REGION Network 10: HMI SpecialFuction Button Control
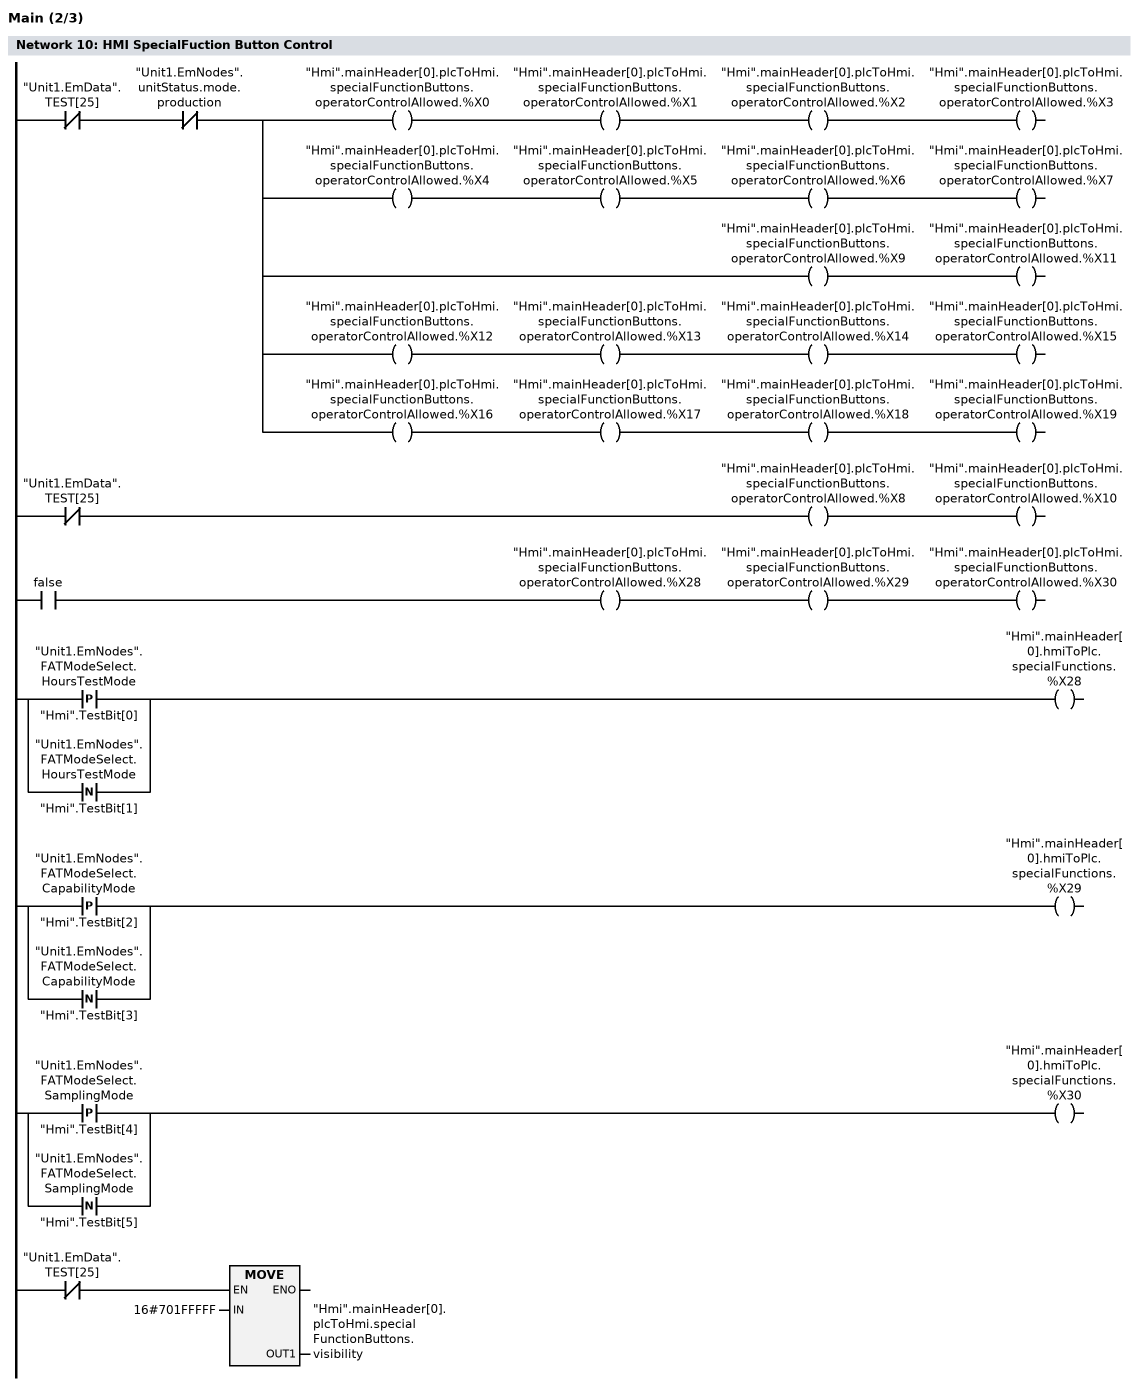
   RUNG wire#powerrail
      I_Contact( "Unit1.EmData".TEST[25] )
      I_Contact( "Unit1.EmNodes".unitStatus.mode.production )
      wire#w1
      Coil( "Hmi".mainHeader[0].plcToHmi.specialFunctionButtons.operatorControlAllowed.%X0 )
      Coil( "Hmi".mainHeader[0].plcToHmi.specialFunctionButtons.operatorControlAllowed.%X1 )
      Coil( "Hmi".mainHeader[0].plcToHmi.specialFunctionButtons.operatorControlAllowed.%X2 )
      Coil( "Hmi".mainHeader[0].plcToHmi.specialFunctionButtons.operatorControlAllowed.%X3 )
   END_RUNG
   RUNG wire#w1
      Coil( "Hmi".mainHeader[0].plcToHmi.specialFunctionButtons.operatorControlAllowed.%X4 )
      Coil( "Hmi".mainHeader[0].plcToHmi.specialFunctionButtons.operatorControlAllowed.%X5 )
      Coil( "Hmi".mainHeader[0].plcToHmi.specialFunctionButtons.operatorControlAllowed.%X6 )
      Coil( "Hmi".mainHeader[0].plcToHmi.specialFunctionButtons.operatorControlAllowed.%X7 )
   END_RUNG
   RUNG wire#w1
      Coil( "Hmi".mainHeader[0].plcToHmi.specialFunctionButtons.operatorControlAllowed.%X9 )
      Coil( "Hmi".mainHeader[0].plcToHmi.specialFunctionButtons.operatorControlAllowed.%X11 )
   END_RUNG
   RUNG wire#w1
      Coil( "Hmi".mainHeader[0].plcToHmi.specialFunctionButtons.operatorControlAllowed.%X12 )
      Coil( "Hmi".mainHeader[0].plcToHmi.specialFunctionButtons.operatorControlAllowed.%X13 )
      Coil( "Hmi".mainHeader[0].plcToHmi.specialFunctionButtons.operatorControlAllowed.%X14 )
      Coil( "Hmi".mainHeader[0].plcToHmi.specialFunctionButtons.operatorControlAllowed.%X15 )
   END_RUNG
   RUNG wire#w1
      Coil( "Hmi".mainHeader[0].plcToHmi.specialFunctionButtons.operatorControlAllowed.%X16 )
      Coil( "Hmi".mainHeader[0].plcToHmi.specialFunctionButtons.operatorControlAllowed.%X17 )
      Coil( "Hmi".mainHeader[0].plcToHmi.specialFunctionButtons.operatorControlAllowed.%X18 )
      Coil( "Hmi".mainHeader[0].plcToHmi.specialFunctionButtons.operatorControlAllowed.%X19 )
   END_RUNG
   RUNG wire#powerrail
      I_Contact( "Unit1.EmData".TEST[25] )
      Coil( "Hmi".mainHeader[0].plcToHmi.specialFunctionButtons.operatorControlAllowed.%X8 )
      Coil( "Hmi".mainHeader[0].plcToHmi.specialFunctionButtons.operatorControlAllowed.%X10 )
   END_RUNG
   RUNG wire#powerrail
      Contact( false )
      Coil( "Hmi".mainHeader[0].plcToHmi.specialFunctionButtons.operatorControlAllowed.%X28 )
      Coil( "Hmi".mainHeader[0].plcToHmi.specialFunctionButtons.operatorControlAllowed.%X29 )
      Coil( "Hmi".mainHeader[0].plcToHmi.specialFunctionButtons.operatorControlAllowed.%X30 )
   END_RUNG
   RUNG wire#powerrail
      P_Contact(operand := "Unit1.EmNodes".FATModeSelect.HoursTestMode, bit := "Hmi".TestBit[0])
      wire#w2
      Coil( "Hmi".mainHeader[0].hmiToPlc.specialFunctions.%X28 )
   END_RUNG
   RUNG wire#powerrail
      N_Contact(operand := "Unit1.EmNodes".FATModeSelect.HoursTestMode, bit := "Hmi".TestBit[1])
   END_RUNG wire#w2
   RUNG wire#powerrail
      P_Contact(operand := "Unit1.EmNodes".FATModeSelect.CapabilityMode, bit := "Hmi".TestBit[2])
      wire#w3
      Coil( "Hmi".mainHeader[0].hmiToPlc.specialFunctions.%X29 )
   END_RUNG
   RUNG wire#powerrail
      N_Contact(operand := "Unit1.EmNodes".FATModeSelect.CapabilityMode, bit := "Hmi".TestBit[3])
   END_RUNG wire#w3
   RUNG wire#powerrail
      P_Contact(operand := "Unit1.EmNodes".FATModeSelect.SamplingMode, bit := "Hmi".TestBit[4])
      wire#w4
      Coil( "Hmi".mainHeader[0].hmiToPlc.specialFunctions.%X30 )
   END_RUNG
   RUNG wire#powerrail
      N_Contact(operand := "Unit1.EmNodes".FATModeSelect.SamplingMode, bit := "Hmi".TestBit[5])
   END_RUNG wire#w4
   RUNG wire#powerrail
      I_Contact( "Unit1.EmData".TEST[25] )
      Move(in := 16#701FFFFF, out1 => "Hmi".mainHeader[0].plcToHmi.specialFunctionButtons.visibility)
   END_RUNG
   // the same network as SCL:
   "Hmi".mainHeader[0].plcToHmi.specialFunctionButtons.operatorControlAllowed.%X0 := NOT "Unit1.EmData".TEST[25] AND NOT "Unit1.EmNodes".unitStatus.mode.production;
   "Hmi".mainHeader[0].plcToHmi.specialFunctionButtons.operatorControlAllowed.%X1 := NOT "Unit1.EmData".TEST[25] AND NOT "Unit1.EmNodes".unitStatus.mode.production;
   "Hmi".mainHeader[0].plcToHmi.specialFunctionButtons.operatorControlAllowed.%X2 := NOT "Unit1.EmData".TEST[25] AND NOT "Unit1.EmNodes".unitStatus.mode.production;
   "Hmi".mainHeader[0].plcToHmi.specialFunctionButtons.operatorControlAllowed.%X3 := NOT "Unit1.EmData".TEST[25] AND NOT "Unit1.EmNodes".unitStatus.mode.production;
   "Hmi".mainHeader[0].plcToHmi.specialFunctionButtons.operatorControlAllowed.%X4 := NOT "Unit1.EmData".TEST[25] AND NOT "Unit1.EmNodes".unitStatus.mode.production;
   "Hmi".mainHeader[0].plcToHmi.specialFunctionButtons.operatorControlAllowed.%X5 := NOT "Unit1.EmData".TEST[25] AND NOT "Unit1.EmNodes".unitStatus.mode.production;
   "Hmi".mainHeader[0].plcToHmi.specialFunctionButtons.operatorControlAllowed.%X6 := NOT "Unit1.EmData".TEST[25] AND NOT "Unit1.EmNodes".unitStatus.mode.production;
   "Hmi".mainHeader[0].plcToHmi.specialFunctionButtons.operatorControlAllowed.%X7 := NOT "Unit1.EmData".TEST[25] AND NOT "Unit1.EmNodes".unitStatus.mode.production;
   "Hmi".mainHeader[0].plcToHmi.specialFunctionButtons.operatorControlAllowed.%X9 := NOT "Unit1.EmData".TEST[25] AND NOT "Unit1.EmNodes".unitStatus.mode.production;
   "Hmi".mainHeader[0].plcToHmi.specialFunctionButtons.operatorControlAllowed.%X11 := NOT "Unit1.EmData".TEST[25] AND NOT "Unit1.EmNodes".unitStatus.mode.production;
   "Hmi".mainHeader[0].plcToHmi.specialFunctionButtons.operatorControlAllowed.%X12 := NOT "Unit1.EmData".TEST[25] AND NOT "Unit1.EmNodes".unitStatus.mode.production;
   "Hmi".mainHeader[0].plcToHmi.specialFunctionButtons.operatorControlAllowed.%X13 := NOT "Unit1.EmData".TEST[25] AND NOT "Unit1.EmNodes".unitStatus.mode.production;
   "Hmi".mainHeader[0].plcToHmi.specialFunctionButtons.operatorControlAllowed.%X14 := NOT "Unit1.EmData".TEST[25] AND NOT "Unit1.EmNodes".unitStatus.mode.production;
   "Hmi".mainHeader[0].plcToHmi.specialFunctionButtons.operatorControlAllowed.%X15 := NOT "Unit1.EmData".TEST[25] AND NOT "Unit1.EmNodes".unitStatus.mode.production;
   "Hmi".mainHeader[0].plcToHmi.specialFunctionButtons.operatorControlAllowed.%X16 := NOT "Unit1.EmData".TEST[25] AND NOT "Unit1.EmNodes".unitStatus.mode.production;
   "Hmi".mainHeader[0].plcToHmi.specialFunctionButtons.operatorControlAllowed.%X17 := NOT "Unit1.EmData".TEST[25] AND NOT "Unit1.EmNodes".unitStatus.mode.production;
   "Hmi".mainHeader[0].plcToHmi.specialFunctionButtons.operatorControlAllowed.%X18 := NOT "Unit1.EmData".TEST[25] AND NOT "Unit1.EmNodes".unitStatus.mode.production;
   "Hmi".mainHeader[0].plcToHmi.specialFunctionButtons.operatorControlAllowed.%X19 := NOT "Unit1.EmData".TEST[25] AND NOT "Unit1.EmNodes".unitStatus.mode.production;
   "Hmi".mainHeader[0].plcToHmi.specialFunctionButtons.operatorControlAllowed.%X8 := NOT "Unit1.EmData".TEST[25];
   "Hmi".mainHeader[0].plcToHmi.specialFunctionButtons.operatorControlAllowed.%X10 := NOT "Unit1.EmData".TEST[25];
   "Hmi".mainHeader[0].plcToHmi.specialFunctionButtons.operatorControlAllowed.%X28 := false;
   "Hmi".mainHeader[0].plcToHmi.specialFunctionButtons.operatorControlAllowed.%X29 := false;
   "Hmi".mainHeader[0].plcToHmi.specialFunctionButtons.operatorControlAllowed.%X30 := false;
   #_w1 := "Unit1.EmNodes".FATModeSelect.HoursTestMode AND NOT "Hmi".TestBit[0];   // rising edge of "Unit1.EmNodes".FATModeSelect.HoursTestMode
   "Hmi".TestBit[0] := "Unit1.EmNodes".FATModeSelect.HoursTestMode;
   #_w2 := NOT "Unit1.EmNodes".FATModeSelect.HoursTestMode AND "Hmi".TestBit[1];   // falling edge of "Unit1.EmNodes".FATModeSelect.HoursTestMode
   "Hmi".TestBit[1] := "Unit1.EmNodes".FATModeSelect.HoursTestMode;
   "Hmi".mainHeader[0].hmiToPlc.specialFunctions.%X28 := #_w1 OR #_w2;
   #_w3 := "Unit1.EmNodes".FATModeSelect.CapabilityMode AND NOT "Hmi".TestBit[2];   // rising edge of "Unit1.EmNodes".FATModeSelect.CapabilityMode
   "Hmi".TestBit[2] := "Unit1.EmNodes".FATModeSelect.CapabilityMode;
   #_w4 := NOT "Unit1.EmNodes".FATModeSelect.CapabilityMode AND "Hmi".TestBit[3];   // falling edge of "Unit1.EmNodes".FATModeSelect.CapabilityMode
   "Hmi".TestBit[3] := "Unit1.EmNodes".FATModeSelect.CapabilityMode;
   "Hmi".mainHeader[0].hmiToPlc.specialFunctions.%X29 := #_w3 OR #_w4;
   #_w5 := "Unit1.EmNodes".FATModeSelect.SamplingMode AND NOT "Hmi".TestBit[4];   // rising edge of "Unit1.EmNodes".FATModeSelect.SamplingMode
   "Hmi".TestBit[4] := "Unit1.EmNodes".FATModeSelect.SamplingMode;
   #_w6 := NOT "Unit1.EmNodes".FATModeSelect.SamplingMode AND "Hmi".TestBit[5];   // falling edge of "Unit1.EmNodes".FATModeSelect.SamplingMode
   "Hmi".TestBit[5] := "Unit1.EmNodes".FATModeSelect.SamplingMode;
   "Hmi".mainHeader[0].hmiToPlc.specialFunctions.%X30 := #_w5 OR #_w6;
   IF NOT "Unit1.EmData".TEST[25] THEN
       "Hmi".mainHeader[0].plcToHmi.specialFunctionButtons.visibility := 16#701FFFFF;
   END_IF;
END_REGION

REGION Network 11
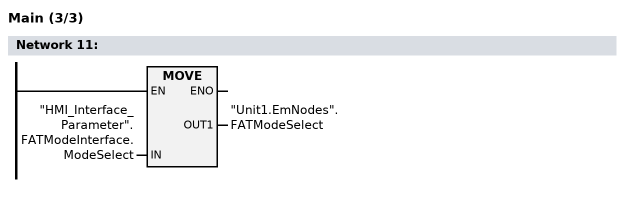
   RUNG wire#powerrail
      Move(in := "HMI_Interface_Parameter".FATModeInterface.ModeSelect, out1 => "Unit1.EmNodes".FATModeSelect)
   END_RUNG
   // the same network as SCL:
   "Unit1.EmNodes".FATModeSelect := "HMI_Interface_Parameter".FATModeInterface.ModeSelect;
END_REGION
END_ORGANIZATION_BLOCK

FUNCTION_BLOCK "CallGlobal"   // FB48, LAD
TITLE = CallGlobal
// All blocks that provide data to the DB Global.Data are called here. That includes blocks to generate system data as well as blocks that connect handle multiple HMIs.
// stored: IsIECCheckEnabled true, MemoryReserve 100, SetENOAutomatically true
   VAR
      statClockSysMemOld { ExternalWritable := 'False'} : Byte;   // Old value system memory evaluation
      statTonTimer : Array[0..10] of IEC_TIMER;
      instLAF_PowerOnOff { ExternalWritable := 'False'} : "LAF_PowerOnOff";
      instLAF_HmiHeaderManager { ExternalWritable := 'False'} : "LAF_HmiHeaderManager";
      instLAF_ClockGen { ExternalWritable := 'False'} : "LAF_ClockGenerator";
      instLSNTP_Server { ExternalWritable := 'False'} : "LSNTP_Server";
      instRemoteAccess { ExternalWritable := 'False'} : "LRemoteAccess_MobilePanelMonitor";
      statPulse : Array[0..99] of Bool;
   END_VAR
   VAR_TEMP
      tempIndex : DInt;   // Temp variable for for loop
      tempAcknowledge : Bool;   // Summarized acknowledge command
      tempPowerOff : Bool;   // Summarized power off command
      tempPowerOn : Bool;   // Summarized power on command
      tempPowerStatus : Int;   // 0 - Off, 1 - Paused, 2 - On
      tempResultXor : Byte;   // Interim result of XOR operation
      tempPosPulse : Byte;   // Interim result puls calculation
   END_VAR
   VAR CONSTANT
      RESET_BUTTON__COULD_BE_ADDED_HERE : Bool := false;   // Placeholder for a potential global reset button
      TRUE : Bool := true;
   END_VAR
   VAR_TEMP   // added for the SCL form of the ladder/FBD networks
      _w1 : Bool;
      _w2 : Bool;
      _w3 : Bool;
   END_VAR
BEGIN

REGION Network 1 (SCL): Summarize HMI commands
   // Read commands for acknowledge, powerOn and powerOff from the different HMI panels and summarize them in temp variables for further logic in this block.
   // Initialize temp variables
   #tempAcknowledge :=
   #tempPowerOff :=
   #tempPowerOn := FALSE;

   // Loop through the HMI panels and summarize the commands
   FOR #tempIndex := 0 TO "NO_OF_PANELS" DO
       #tempAcknowledge := #tempAcknowledge OR "Hmi".mainHeader[#tempIndex].hmiToPlc.acknowledge;
       #tempPowerOff := #tempPowerOff OR "Hmi".mainHeader[#tempIndex].hmiToPlc.powerCommands.%X0;
       #tempPowerOn := #tempPowerOn OR "Hmi".mainHeader[#tempIndex].hmiToPlc.powerCommands.%X1;
   END_FOR;
END_REGION

REGION Network 2: Global Acknowledge
   // The global acknowledge command from the hmi button is assigned to Global.Data.general.acknowledge: This bit it forwarded to all underlaying modules
   // If a hard-wired global reset button exists, it can
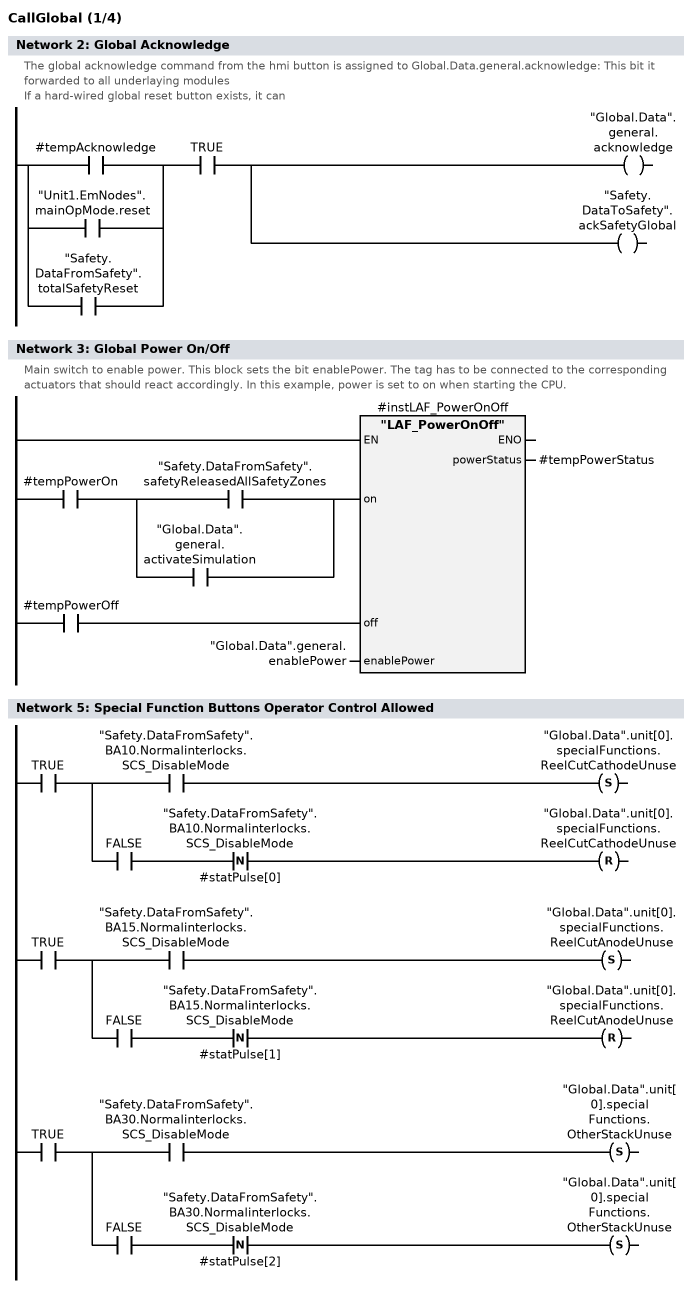
   RUNG wire#powerrail
      Contact( #tempAcknowledge )
      wire#w1
      Contact( TRUE )
      wire#w2
      Coil( "Global.Data".general.acknowledge )
   END_RUNG
   RUNG wire#powerrail
      Contact( "Unit1.EmNodes".mainOpMode.reset )
   END_RUNG wire#w1
   RUNG wire#powerrail
      Contact( "Safety.DataFromSafety".totalSafetyReset )
   END_RUNG wire#w1
   RUNG wire#w2
      Coil( "Safety.DataToSafety".ackSafetyGlobal )
   END_RUNG
   // the same network as SCL:
   "Global.Data".general.acknowledge := (#tempAcknowledge OR "Unit1.EmNodes".mainOpMode.reset OR "Safety.DataFromSafety".totalSafetyReset) AND TRUE;
   "Safety.DataToSafety".ackSafetyGlobal := "Global.Data".general.acknowledge;
END_REGION

REGION Network 3: Global Power On/Off
   // Main switch to enable power. This block sets the bit enablePower. The tag has to be connected to the corresponding actuators that should react accordingly. In this example, power is set to on when starting the CPU.
   RUNG wire#powerrail
      #instLAF_PowerOnOff(on := wire#w2, off := wire#w3, enablePower := "Global.Data".general.enablePower, powerStatus => #tempPowerStatus)
   END_RUNG
   RUNG wire#powerrail
      Contact( #tempPowerOn )
      wire#w1
      Contact( "Safety.DataFromSafety".safetyReleasedAllSafetyZones )
   END_RUNG wire#w2
   RUNG wire#w1
      Contact( "Global.Data".general.activateSimulation )
   END_RUNG wire#w2
   RUNG wire#powerrail
      Contact( #tempPowerOff )
   END_RUNG wire#w3
   // the same network as SCL:
   #instLAF_PowerOnOff(on := #tempPowerOn AND ("Safety.DataFromSafety".safetyReleasedAllSafetyZones OR "Global.Data".general.activateSimulation),   // "LAF_PowerOnOff"
                       off := #tempPowerOff,
                       enablePower := "Global.Data".general.enablePower,
                       powerStatus => #tempPowerStatus);
END_REGION

REGION Network 4 (SCL): Write power status to HMI panels
   // Write power status back to all connected HMI panels
   // Loop through the panels and set the power status
   FOR #tempIndex := 0 TO "NO_OF_PANELS" DO
       "Hmi".mainHeader[#tempIndex].plcToHmi.powerStatus := #tempPowerStatus;
   END_FOR;
END_REGION

REGION Network 5: Special Function Buttons Operator Control Allowed
   RUNG wire#powerrail
      Contact( TRUE )
      wire#w1
      Contact( "Safety.DataFromSafety".BA10.Normalinterlocks.SCS_DisableMode )
      S_Coil( "Global.Data".unit[0].specialFunctions.ReelCutCathodeUnuse )
   END_RUNG
   RUNG wire#w1
      Contact( FALSE )
      N_Contact(operand := "Safety.DataFromSafety".BA10.Normalinterlocks.SCS_DisableMode, bit := #statPulse[0])
      R_Coil( "Global.Data".unit[0].specialFunctions.ReelCutCathodeUnuse )
   END_RUNG
   RUNG wire#powerrail
      Contact( TRUE )
      wire#w2
      Contact( "Safety.DataFromSafety".BA15.Normalinterlocks.SCS_DisableMode )
      S_Coil( "Global.Data".unit[0].specialFunctions.ReelCutAnodeUnuse )
   END_RUNG
   RUNG wire#w2
      Contact( FALSE )
      N_Contact(operand := "Safety.DataFromSafety".BA15.Normalinterlocks.SCS_DisableMode, bit := #statPulse[1])
      R_Coil( "Global.Data".unit[0].specialFunctions.ReelCutAnodeUnuse )
   END_RUNG
   RUNG wire#powerrail
      Contact( TRUE )
      wire#w3
      Contact( "Safety.DataFromSafety".BA30.Normalinterlocks.SCS_DisableMode )
      S_Coil( "Global.Data".unit[0].specialFunctions.OtherStackUnuse )
   END_RUNG
   RUNG wire#w3
      Contact( FALSE )
      N_Contact(operand := "Safety.DataFromSafety".BA30.Normalinterlocks.SCS_DisableMode, bit := #statPulse[2])
      S_Coil( "Global.Data".unit[0].specialFunctions.OtherStackUnuse )
   END_RUNG
   // the same network as SCL:
   IF TRUE AND "Safety.DataFromSafety".BA10.Normalinterlocks.SCS_DisableMode THEN
       "Global.Data".unit[0].specialFunctions.ReelCutCathodeUnuse := TRUE;
   END_IF;
   #_w1 := TRUE AND FALSE AND NOT "Safety.DataFromSafety".BA10.Normalinterlocks.SCS_DisableMode AND #statPulse[0];   // falling edge of "Safety.DataFromSafety".BA10.Normalinterlocks.SCS_DisableMode
   #statPulse[0] := "Safety.DataFromSafety".BA10.Normalinterlocks.SCS_DisableMode;
   IF #_w1 THEN "Global.Data".unit[0].specialFunctions.ReelCutCathodeUnuse := FALSE; END_IF;
   IF TRUE AND "Safety.DataFromSafety".BA15.Normalinterlocks.SCS_DisableMode THEN
       "Global.Data".unit[0].specialFunctions.ReelCutAnodeUnuse := TRUE;
   END_IF;
   #_w2 := TRUE AND FALSE AND NOT "Safety.DataFromSafety".BA15.Normalinterlocks.SCS_DisableMode AND #statPulse[1];   // falling edge of "Safety.DataFromSafety".BA15.Normalinterlocks.SCS_DisableMode
   #statPulse[1] := "Safety.DataFromSafety".BA15.Normalinterlocks.SCS_DisableMode;
   IF #_w2 THEN "Global.Data".unit[0].specialFunctions.ReelCutAnodeUnuse := FALSE; END_IF;
   IF TRUE AND "Safety.DataFromSafety".BA30.Normalinterlocks.SCS_DisableMode THEN
       "Global.Data".unit[0].specialFunctions.OtherStackUnuse := TRUE;
   END_IF;
   #_w3 := TRUE AND FALSE AND NOT "Safety.DataFromSafety".BA30.Normalinterlocks.SCS_DisableMode AND #statPulse[2];   // falling edge of "Safety.DataFromSafety".BA30.Normalinterlocks.SCS_DisableMode
   #statPulse[2] := "Safety.DataFromSafety".BA30.Normalinterlocks.SCS_DisableMode;
   IF #_w3 THEN "Global.Data".unit[0].specialFunctions.OtherStackUnuse := TRUE; END_IF;
END_REGION

REGION Network 6: HMI Control Header
   // Read the input from the control header in the HMI an distribute information to the according units. Vice versa, summarize the unit information and provide it to the control header to display e.g. the modes and states.
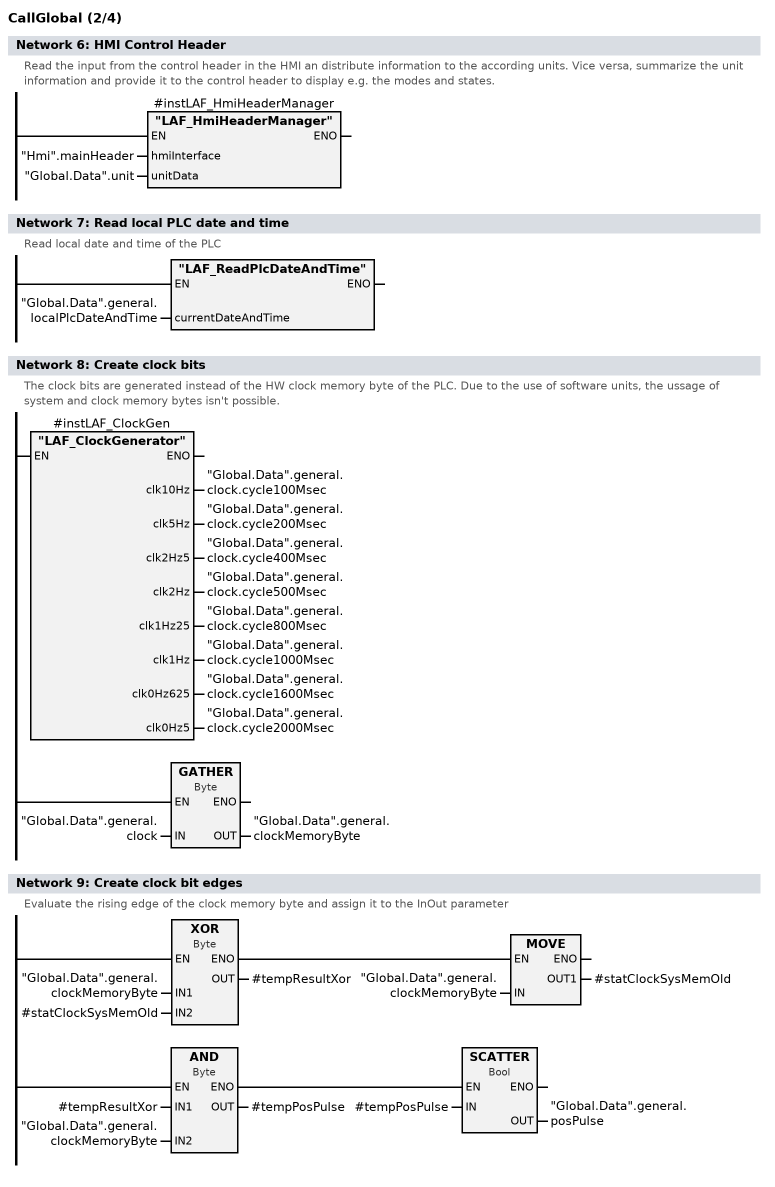
   RUNG wire#powerrail
      #instLAF_HmiHeaderManager(hmiInterface := "Hmi".mainHeader, unitData := "Global.Data".unit)
   END_RUNG
   // the same network as SCL:
   #instLAF_HmiHeaderManager(hmiInterface := "Hmi".mainHeader, unitData := "Global.Data".unit);   // "LAF_HmiHeaderManager"
END_REGION

REGION Network 7: Read local PLC date and time
   // Read local date and time of the PLC
   RUNG wire#powerrail
      "LAF_ReadPlcDateAndTime"(currentDateAndTime := "Global.Data".general.localPlcDateAndTime)
   END_RUNG
   // the same network as SCL:
   "LAF_ReadPlcDateAndTime"(currentDateAndTime := "Global.Data".general.localPlcDateAndTime);
END_REGION

REGION Network 8: Create clock bits
   // The clock bits are generated instead of the HW clock memory byte of the PLC. Due to the use of software units, the ussage of system and clock memory bytes isn't possible.
   RUNG wire#powerrail
      #instLAF_ClockGen(clk10Hz => "Global.Data".general.clock.cycle100Msec, clk5Hz => "Global.Data".general.clock.cycle200Msec, clk2Hz5 => "Global.Data".general.clock.cycle400Msec, clk2Hz => "Global.Data".general.clock.cycle500Msec, clk1Hz25 => "Global.Data".general.clock.cycle800Msec, clk1Hz => "Global.Data".general.clock.cycle1000Msec, clk0Hz625 => "Global.Data".general.clock.cycle1600Msec, clk0Hz5 => "Global.Data".general.clock.cycle2000Msec)
   END_RUNG
   RUNG wire#powerrail
      { S7_Templates := "[dest_type := Byte, src_type := Bool]" } GATHER(IN := "Global.Data".general.clock, OUT => "Global.Data".general.clockMemoryByte)
   END_RUNG
   // the same network as SCL:
   #instLAF_ClockGen(clk10Hz => "Global.Data".general.clock.cycle100Msec,   // "LAF_ClockGenerator"
                     clk5Hz => "Global.Data".general.clock.cycle200Msec,
                     clk2Hz5 => "Global.Data".general.clock.cycle400Msec,
                     clk2Hz => "Global.Data".general.clock.cycle500Msec,
                     clk1Hz25 => "Global.Data".general.clock.cycle800Msec,
                     clk1Hz => "Global.Data".general.clock.cycle1000Msec,
                     clk0Hz625 => "Global.Data".general.clock.cycle1600Msec,
                     clk0Hz5 => "Global.Data".general.clock.cycle2000Msec);
   GATHER(IN := "Global.Data".general.clock, OUT => "Global.Data".general.clockMemoryByte);
END_REGION

REGION Network 9: Create clock bit edges
   // Evaluate the rising edge of the clock memory byte and assign it to the InOut parameter
   #tempResultXor := "Global.Data".general.clockMemoryByte XOR #statClockSysMemOld;
   #statClockSysMemOld := "Global.Data".general.clockMemoryByte;
   #tempPosPulse := #tempResultXor AND "Global.Data".general.clockMemoryByte;
   SCATTER(IN := #tempPosPulse, OUT => "Global.Data".general.posPulse);
END_REGION

REGION Network 10: Time Synchronisation (NTP)
   // With the LSNTP_Server block, the NTP server will be enabled on S7 PLC, to wich the NTP client (e.g. Panel), can synchronize their data and time.
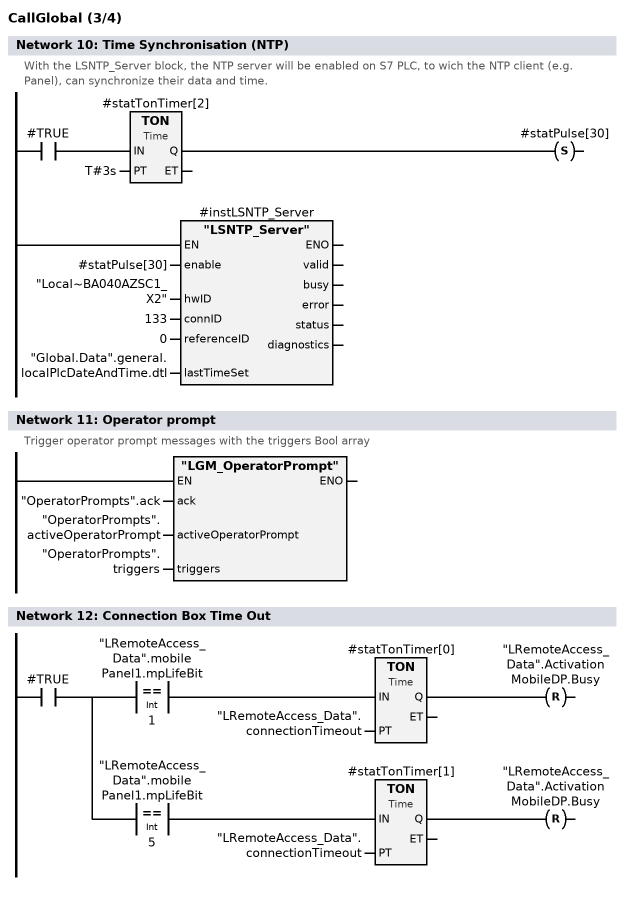
   RUNG wire#powerrail
      Contact( #TRUE )
      { S7_Templates := "time_type := Time" } #statTonTimer[2].TON(pt := T#3s, et =>)
      S_Coil( #statPulse[30] )
   END_RUNG
   RUNG wire#powerrail
      #instLSNTP_Server(enable := #statPulse[30], hwID := "Local~BA040AZSC1_X2", connID := 133, referenceID := 0, lastTimeSet := "Global.Data".general.localPlcDateAndTime.dtl, valid =>, busy =>, error =>, status =>, diagnostics =>)
   END_RUNG
   // the same network as SCL:
   #statTonTimer[2].TON(IN := #TRUE, PT := T#3s);
   IF #statTonTimer[2].Q THEN #statPulse[30] := TRUE; END_IF;
   #instLSNTP_Server(enable := #statPulse[30],   // "LSNTP_Server"
                     hwID := "Local~BA040AZSC1_X2",
                     connID := 133,
                     referenceID := 0,
                     lastTimeSet := "Global.Data".general.localPlcDateAndTime.dtl);
END_REGION

REGION Network 11: Operator prompt
   // Trigger operator prompt messages with the triggers Bool array
   RUNG wire#powerrail
      "LGM_OperatorPrompt"(ack := "OperatorPrompts".ack, activeOperatorPrompt := "OperatorPrompts".activeOperatorPrompt, triggers := "OperatorPrompts".triggers)
   END_RUNG
   // the same network as SCL:
   "LGM_OperatorPrompt"(ack := "OperatorPrompts".ack,
                        activeOperatorPrompt := "OperatorPrompts".activeOperatorPrompt,
                        triggers := "OperatorPrompts".triggers);
END_REGION

REGION Network 12: Connection Box Time Out
   RUNG wire#powerrail
      Contact( #TRUE )
      wire#w1
      { S7_Templates := "SrcType := Int" } EQ_Contact(in1 := "LRemoteAccess_Data".mobilePanel1.mpLifeBit, in2 := 1)
      { S7_Templates := "time_type := Time" } #statTonTimer[0].TON(pt := "LRemoteAccess_Data".connectionTimeout, et =>)
      R_Coil( "LRemoteAccess_Data".ActivationMobileDP.Busy )
   END_RUNG
   RUNG wire#w1
      { S7_Templates := "SrcType := Int" } EQ_Contact(in1 := "LRemoteAccess_Data".mobilePanel1.mpLifeBit, in2 := 5)
      { S7_Templates := "time_type := Time" } #statTonTimer[1].TON(pt := "LRemoteAccess_Data".connectionTimeout, et =>)
      R_Coil( "LRemoteAccess_Data".ActivationMobileDP.Busy )
   END_RUNG
   // the same network as SCL:
   #statTonTimer[0].TON(IN := #TRUE AND ("LRemoteAccess_Data".mobilePanel1.mpLifeBit = 1),
                        PT := "LRemoteAccess_Data".connectionTimeout);
   IF #statTonTimer[0].Q THEN "LRemoteAccess_Data".ActivationMobileDP.Busy := FALSE; END_IF;
   #statTonTimer[1].TON(IN := #TRUE AND ("LRemoteAccess_Data".mobilePanel1.mpLifeBit = 5),
                        PT := "LRemoteAccess_Data".connectionTimeout);
   IF #statTonTimer[1].Q THEN "LRemoteAccess_Data".ActivationMobileDP.Busy := FALSE; END_IF;
END_REGION

REGION Network 13: Connection box is connected
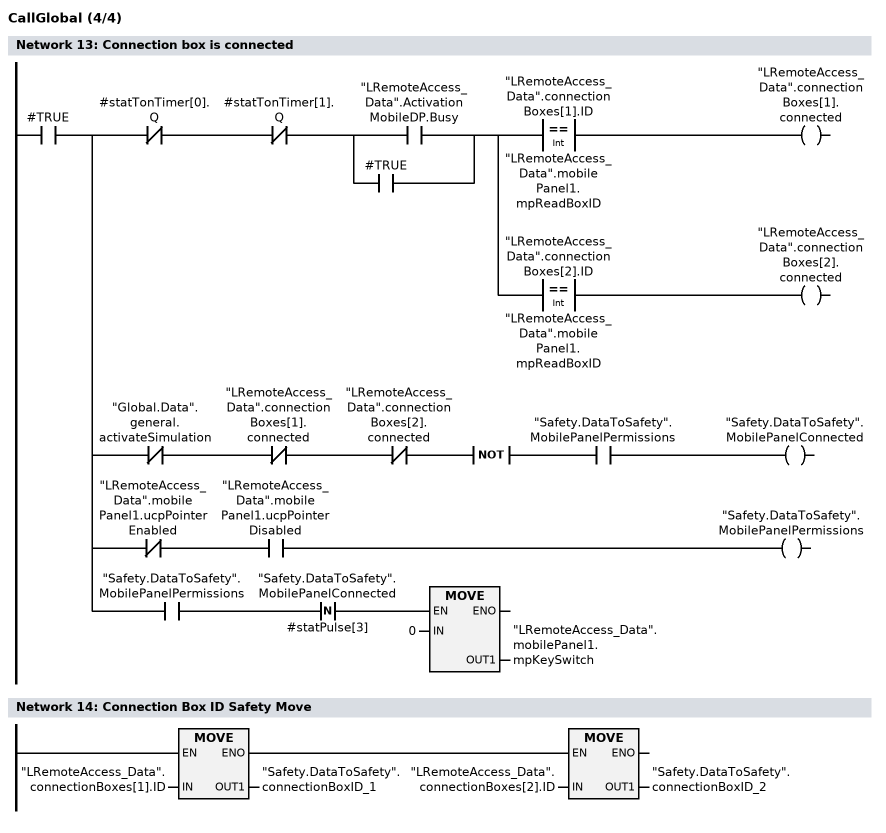
   RUNG wire#powerrail
      Contact( #TRUE )
      wire#w1
      I_Contact( #statTonTimer[0].Q )
      I_Contact( #statTonTimer[1].Q )
      wire#w2
      Contact( "LRemoteAccess_Data".ActivationMobileDP.Busy )
      wire#w3
      { S7_Templates := "SrcType := Int" } EQ_Contact(in1 := "LRemoteAccess_Data".connectionBoxes[1].ID, in2 := "LRemoteAccess_Data".mobilePanel1.mpReadBoxID)
      Coil( "LRemoteAccess_Data".connectionBoxes[1].connected )
   END_RUNG
   RUNG wire#w2
      Contact( #TRUE )
   END_RUNG wire#w3
   RUNG wire#w3
      { S7_Templates := "SrcType := Int" } EQ_Contact(in1 := "LRemoteAccess_Data".connectionBoxes[2].ID, in2 := "LRemoteAccess_Data".mobilePanel1.mpReadBoxID)
      Coil( "LRemoteAccess_Data".connectionBoxes[2].connected )
   END_RUNG
   RUNG wire#w1
      I_Contact( "Global.Data".general.activateSimulation )
      I_Contact( "LRemoteAccess_Data".connectionBoxes[1].connected )
      I_Contact( "LRemoteAccess_Data".connectionBoxes[2].connected )
      Not()
      Contact( "Safety.DataToSafety".MobilePanelPermissions )
      Coil( "Safety.DataToSafety".MobilePanelConnected )
   END_RUNG
   RUNG wire#w1
      I_Contact( "LRemoteAccess_Data".mobilePanel1.ucpPointerEnabled )
      Contact( "LRemoteAccess_Data".mobilePanel1.ucpPointerDisabled )
      Coil( "Safety.DataToSafety".MobilePanelPermissions )
   END_RUNG
   RUNG wire#w1
      Contact( "Safety.DataToSafety".MobilePanelPermissions )
      N_Contact(operand := "Safety.DataToSafety".MobilePanelConnected, bit := #statPulse[3])
      Move(in := 0, out1 => "LRemoteAccess_Data".mobilePanel1.mpKeySwitch)
   END_RUNG
   // the same network as SCL:
   #_w1 := #TRUE AND NOT #statTonTimer[0].Q AND NOT #statTonTimer[1].Q AND ("LRemoteAccess_Data".ActivationMobileDP.Busy OR #TRUE);
   "LRemoteAccess_Data".connectionBoxes[1].connected := #_w1 AND ("LRemoteAccess_Data".connectionBoxes[1].ID = "LRemoteAccess_Data".mobilePanel1.mpReadBoxID);
   "LRemoteAccess_Data".connectionBoxes[2].connected := #_w1 AND ("LRemoteAccess_Data".connectionBoxes[2].ID = "LRemoteAccess_Data".mobilePanel1.mpReadBoxID);
   "Safety.DataToSafety".MobilePanelConnected := NOT (#TRUE AND NOT "Global.Data".general.activateSimulation AND NOT "LRemoteAccess_Data".connectionBoxes[1].connected AND NOT "LRemoteAccess_Data".connectionBoxes[2].connected) AND "Safety.DataToSafety".MobilePanelPermissions;
   "Safety.DataToSafety".MobilePanelPermissions := #TRUE AND NOT "LRemoteAccess_Data".mobilePanel1.ucpPointerEnabled AND "LRemoteAccess_Data".mobilePanel1.ucpPointerDisabled;
   #_w2 := #TRUE AND "Safety.DataToSafety".MobilePanelPermissions AND NOT "Safety.DataToSafety".MobilePanelConnected AND #statPulse[3];   // falling edge of "Safety.DataToSafety".MobilePanelConnected
   #statPulse[3] := "Safety.DataToSafety".MobilePanelConnected;
   IF #_w2 THEN "LRemoteAccess_Data".mobilePanel1.mpKeySwitch := 0; END_IF;
END_REGION

REGION Network 14: Connection Box ID Safety Move
   RUNG wire#powerrail
      Move(in := "LRemoteAccess_Data".connectionBoxes[1].ID, out1 => "Safety.DataToSafety".connectionBoxID_1)
      Move(in := "LRemoteAccess_Data".connectionBoxes[2].ID, out1 => "Safety.DataToSafety".connectionBoxID_2)
   END_RUNG
   // the same network as SCL:
   "Safety.DataToSafety".connectionBoxID_1 := "LRemoteAccess_Data".connectionBoxes[1].ID;
   "Safety.DataToSafety".connectionBoxID_2 := "LRemoteAccess_Data".connectionBoxes[2].ID;
END_REGION
END_FUNCTION_BLOCK

FUNCTION_BLOCK "CallSimulation"   // FB19, LAD
// stored: MemoryReserve 100, SetENOAutomatically false
   VAR
      instSimRotaryAxis { ExternalAccessible := 'False'; ExternalVisible := 'False'; ExternalWritable := 'False'} : Array[0..49] of "LER_SimHmiRotaryAxis";
      Unwindwe1 { S7_SetPoint := 'True'} : "LER_SimHmiRotaryAxis";
      IEC_Timer_0_Instance { S7_SetPoint := 'True'} : TON_TIME;
      "LER_SimAxis+_Axis07_pnp1X" { S7_SetPoint := 'True'} : "LER_SimAxis+";
      "LER_SimAxis+_Axis10_pnp1Z" { S7_SetPoint := 'True'} : "LER_SimAxis+";
      "LER_SimAxis+_Axis8_pnp2X" { S7_SetPoint := 'True'} : "LER_SimAxis+";
      "LER_SimAxis+_Axis13_pnp2Z" { S7_SetPoint := 'True'} : "LER_SimAxis+";
      "LER_SimAxis+_Axis12_pnp1Z" { S7_SetPoint := 'True'} : "LER_SimAxis+";
      "LER_SimAxis+_Axis14_pnp2Z" { S7_SetPoint := 'True'} : "LER_SimAxis+";
      "LER_SimAxis+_Axis34_cutterX" { S7_SetPoint := 'True'} : "LER_SimAxis+";
      "LER_SimAxis+_Axis35_cutterZ" { S7_SetPoint := 'True'} : "LER_SimAxis+";
      "LER_SimAxis-_Axis36_GripperX" { S7_SetPoint := 'True'} : "LER_SimAxis-";
      "LER_SimAxis+_Axis37_gripperZ" { S7_SetPoint := 'True'} : "LER_SimAxis+";
      "LER_SimAxis-_Axis32_StackTableZ" { S7_SetPoint := 'True'} : "LER_SimAxis-";
      "LER_SimAxis+_Axis21_roller" { S7_SetPoint := 'True'} : "LER_SimAxis+";
      "LER_SimAxis+_gripperAxis_C" { S7_SetPoint := 'True'} : "LER_SimAxis+";
      IEC_Timer_1_Instance { S7_SetPoint := 'True'} : TON_TIME;
      "LER_SimAxis+_Axis05_pnp1X" { S7_SetPoint := 'True'} : "LER_SimAxis+";
      "LER_SimAxis+_Axis06_pnp2X" { S7_SetPoint := 'True'} : "LER_SimAxis+";
   END_VAR
   VAR CONSTANT
      FALSE : Bool := FALSE;
      TRUE : Bool := TRUE;
   END_VAR
   VAR_TEMP   // added for the SCL form of the ladder/FBD networks
      _w1 : Bool;
      _w2 : Bool;
      _w3 : Bool;
      _w4 : Bool;
      _w5 : Bool;
      _w6 : Bool;
      _w7 : Bool;
      _w8 : Bool;
   END_VAR
BEGIN

REGION Network 1: SIMIT simulation currently running
   // The input "0.000CC1-KE50_I1.6_SimitRunning" is a life bit from SIMIT, which is always TRUE while SIMIT is running. The following actions are performed in that case:
   // - Simulation button in HMI is not shown when a SIMIT simulation is currently running
   // - Deactivate PLC internal simulation while SIMIT simulation is running
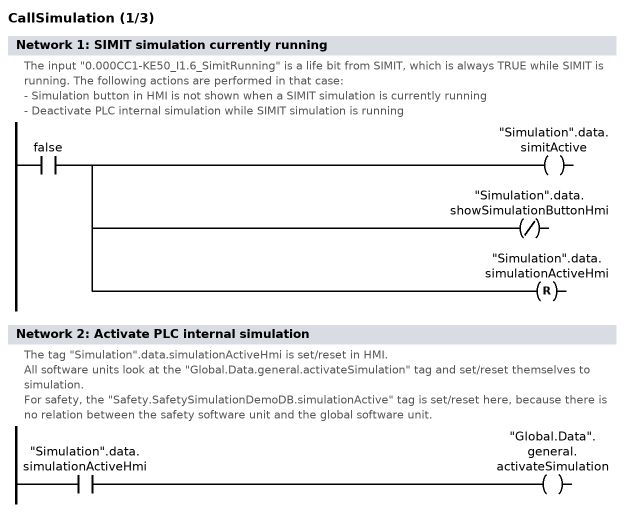
   RUNG wire#powerrail
      Contact( false )
      wire#w1
      Coil( "Simulation".data.simitActive )
   END_RUNG
   RUNG wire#w1
      I_Coil( "Simulation".data.showSimulationButtonHmi )
   END_RUNG
   RUNG wire#w1
      R_Coil( "Simulation".data.simulationActiveHmi )
   END_RUNG
   // the same network as SCL:
   "Simulation".data.simitActive := false;
   "Simulation".data.showSimulationButtonHmi := NOT false;
   IF false THEN "Simulation".data.simulationActiveHmi := FALSE; END_IF;
END_REGION

REGION Network 2: Activate PLC internal simulation
   // The tag "Simulation".data.simulationActiveHmi is set/reset in HMI.
   // 
   // All software units look at the "Global.Data.general.activateSimulation" tag and set/reset themselves to simulation.
   // 
   // For safety, the "Safety.SafetySimulationDemoDB.simulationActive" tag is set/reset here, because there is no relation between the safety software unit and the global software unit.
   RUNG wire#powerrail
      Contact( "Simulation".data.simulationActiveHmi )
      Coil( "Global.Data".general.activateSimulation )
   END_RUNG
   // the same network as SCL:
   "Global.Data".general.activateSimulation := "Simulation".data.simulationActiveHmi;
END_REGION

REGION Network 3: Simulation Linear Axis
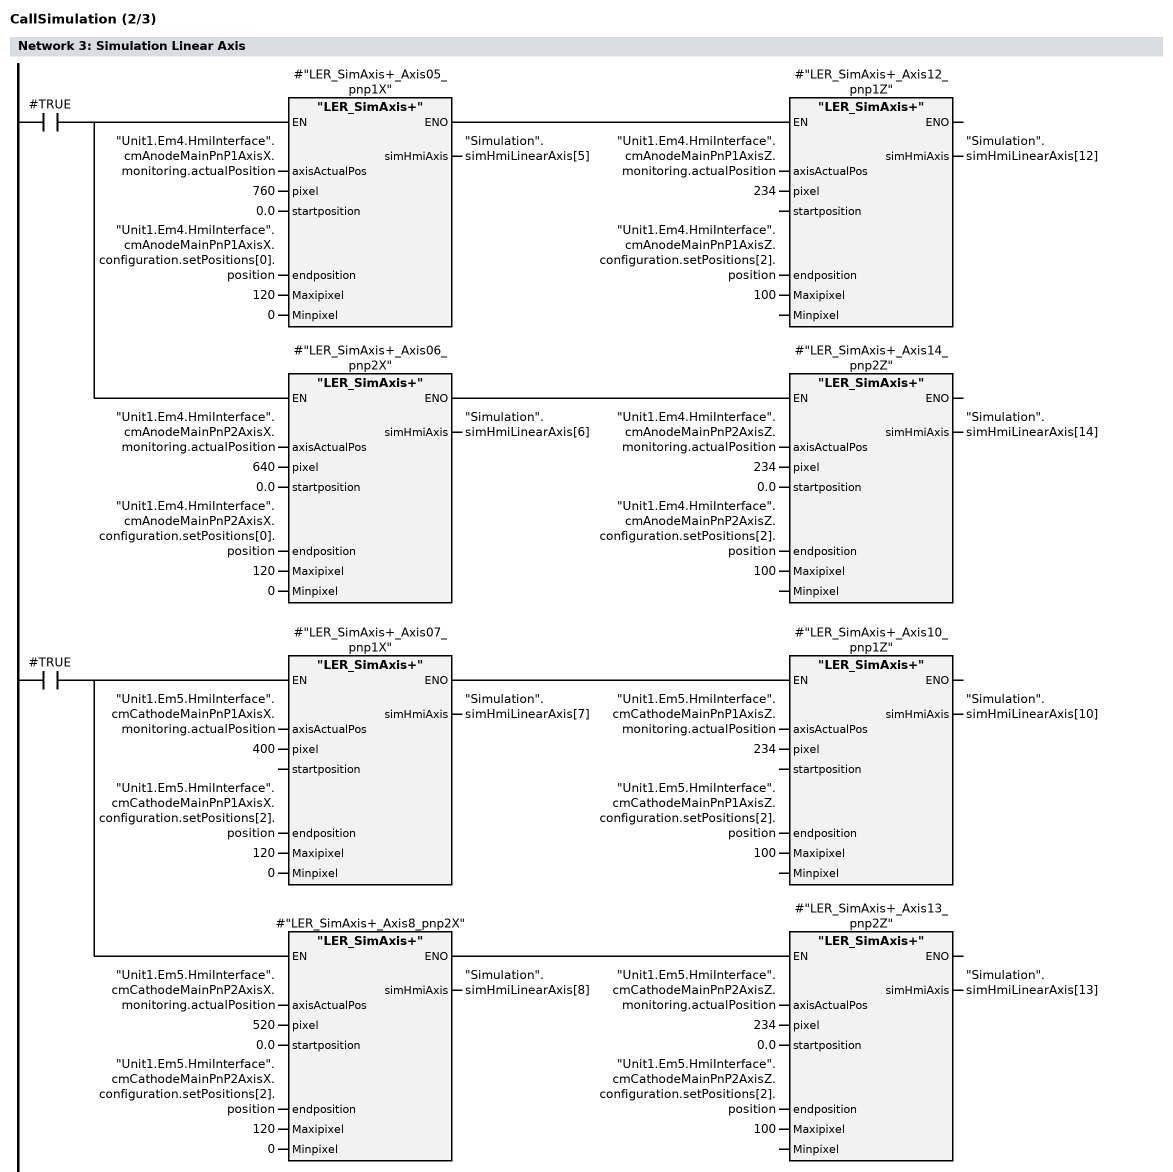
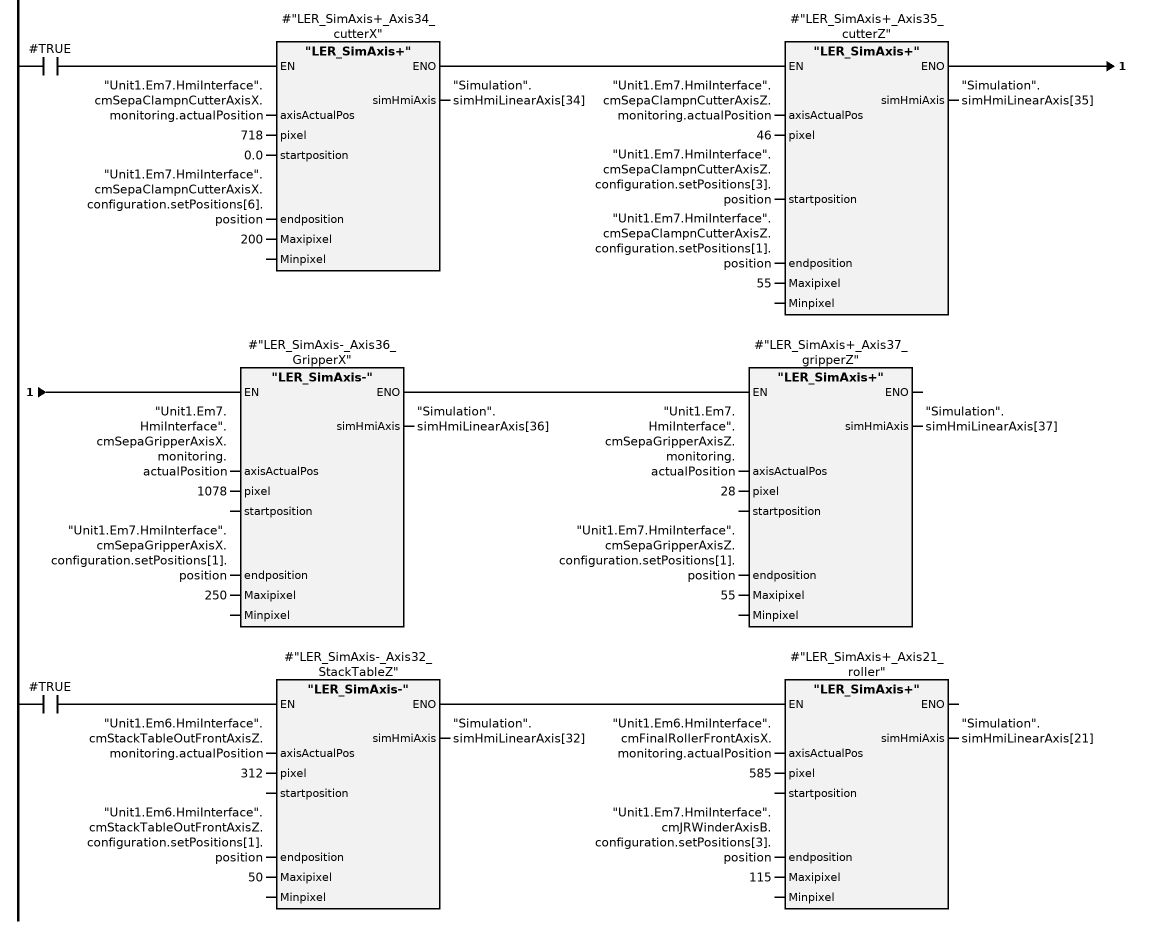
   RUNG wire#powerrail
      Contact( #TRUE )
      wire#w1
      #"LER_SimAxis+_Axis05_pnp1X"(axisActualPos := "Unit1.Em4.HmiInterface".cmAnodeMainPnP1AxisX.monitoring.actualPosition, pixel := 760, startposition := 0.0, endposition := "Unit1.Em4.HmiInterface".cmAnodeMainPnP1AxisX.configuration.setPositions[0].position, Maxipixel := 120, Minpixel := 0, simHmiAxis => "Simulation".simHmiLinearAxis[5])
      #"LER_SimAxis+_Axis12_pnp1Z"(axisActualPos := "Unit1.Em4.HmiInterface".cmAnodeMainPnP1AxisZ.monitoring.actualPosition, pixel := 234, startposition :=, endposition := "Unit1.Em4.HmiInterface".cmAnodeMainPnP1AxisZ.configuration.setPositions[2].position, Maxipixel := 100, Minpixel :=, simHmiAxis => "Simulation".simHmiLinearAxis[12])
   END_RUNG
   RUNG wire#w1
      #"LER_SimAxis+_Axis06_pnp2X"(axisActualPos := "Unit1.Em4.HmiInterface".cmAnodeMainPnP2AxisX.monitoring.actualPosition, pixel := 640, startposition := 0.0, endposition := "Unit1.Em4.HmiInterface".cmAnodeMainPnP2AxisX.configuration.setPositions[0].position, Maxipixel := 120, Minpixel := 0, simHmiAxis => "Simulation".simHmiLinearAxis[6])
      #"LER_SimAxis+_Axis14_pnp2Z"(axisActualPos := "Unit1.Em4.HmiInterface".cmAnodeMainPnP2AxisZ.monitoring.actualPosition, pixel := 234, startposition := 0.0, endposition := "Unit1.Em4.HmiInterface".cmAnodeMainPnP2AxisZ.configuration.setPositions[2].position, Maxipixel := 100, Minpixel :=, simHmiAxis => "Simulation".simHmiLinearAxis[14])
   END_RUNG
   RUNG wire#powerrail
      Contact( #TRUE )
      wire#w2
      #"LER_SimAxis+_Axis07_pnp1X"(axisActualPos := "Unit1.Em5.HmiInterface".cmCathodeMainPnP1AxisX.monitoring.actualPosition, pixel := 400, startposition :=, endposition := "Unit1.Em5.HmiInterface".cmCathodeMainPnP1AxisX.configuration.setPositions[2].position, Maxipixel := 120, Minpixel := 0, simHmiAxis => "Simulation".simHmiLinearAxis[7])
      #"LER_SimAxis+_Axis10_pnp1Z"(axisActualPos := "Unit1.Em5.HmiInterface".cmCathodeMainPnP1AxisZ.monitoring.actualPosition, pixel := 234, startposition :=, endposition := "Unit1.Em5.HmiInterface".cmCathodeMainPnP1AxisZ.configuration.setPositions[2].position, Maxipixel := 100, Minpixel :=, simHmiAxis => "Simulation".simHmiLinearAxis[10])
   END_RUNG
   RUNG wire#w2
      #"LER_SimAxis+_Axis8_pnp2X"(axisActualPos := "Unit1.Em5.HmiInterface".cmCathodeMainPnP2AxisX.monitoring.actualPosition, pixel := 520, startposition := 0.0, endposition := "Unit1.Em5.HmiInterface".cmCathodeMainPnP2AxisX.configuration.setPositions[2].position, Maxipixel := 120, Minpixel := 0, simHmiAxis => "Simulation".simHmiLinearAxis[8])
      #"LER_SimAxis+_Axis13_pnp2Z"(axisActualPos := "Unit1.Em5.HmiInterface".cmCathodeMainPnP2AxisZ.monitoring.actualPosition, pixel := 234, startposition := 0.0, endposition := "Unit1.Em5.HmiInterface".cmCathodeMainPnP2AxisZ.configuration.setPositions[2].position, Maxipixel := 100, Minpixel :=, simHmiAxis => "Simulation".simHmiLinearAxis[13])
   END_RUNG
   RUNG wire#powerrail
      Contact( #TRUE )
      #"LER_SimAxis+_Axis34_cutterX"(axisActualPos := "Unit1.Em7.HmiInterface".cmSepaClampnCutterAxisX.monitoring.actualPosition, pixel := 718, startposition := 0.0, endposition := "Unit1.Em7.HmiInterface".cmSepaClampnCutterAxisX.configuration.setPositions[6].position, Maxipixel := 200, Minpixel :=, simHmiAxis => "Simulation".simHmiLinearAxis[34])
      #"LER_SimAxis+_Axis35_cutterZ"(axisActualPos := "Unit1.Em7.HmiInterface".cmSepaClampnCutterAxisZ.monitoring.actualPosition, pixel := 46, startposition := "Unit1.Em7.HmiInterface".cmSepaClampnCutterAxisZ.configuration.setPositions[3].position, endposition := "Unit1.Em7.HmiInterface".cmSepaClampnCutterAxisZ.configuration.setPositions[1].position, Maxipixel := 55, Minpixel :=, simHmiAxis => "Simulation".simHmiLinearAxis[35])
      #"LER_SimAxis-_Axis36_GripperX"(axisActualPos := "Unit1.Em7.HmiInterface".cmSepaGripperAxisX.monitoring.actualPosition, pixel := 1078, startposition :=, endposition := "Unit1.Em7.HmiInterface".cmSepaGripperAxisX.configuration.setPositions[1].position, Maxipixel := 250, Minpixel :=, simHmiAxis => "Simulation".simHmiLinearAxis[36])
      #"LER_SimAxis+_Axis37_gripperZ"(axisActualPos := "Unit1.Em7.HmiInterface".cmSepaGripperAxisZ.monitoring.actualPosition, pixel := 28, startposition :=, endposition := "Unit1.Em7.HmiInterface".cmSepaGripperAxisZ.configuration.setPositions[1].position, Maxipixel := 55, Minpixel :=, simHmiAxis => "Simulation".simHmiLinearAxis[37])
   END_RUNG
   RUNG wire#powerrail
      Contact( #TRUE )
      #"LER_SimAxis-_Axis32_StackTableZ"(axisActualPos := "Unit1.Em6.HmiInterface".cmStackTableOutFrontAxisZ.monitoring.actualPosition, pixel := 312, startposition :=, endposition := "Unit1.Em6.HmiInterface".cmStackTableOutFrontAxisZ.configuration.setPositions[1].position, Maxipixel := 50, Minpixel :=, simHmiAxis => "Simulation".simHmiLinearAxis[32])
      #"LER_SimAxis+_Axis21_roller"(axisActualPos := "Unit1.Em6.HmiInterface".cmFinalRollerFrontAxisX.monitoring.actualPosition, pixel := 585, startposition :=, endposition := "Unit1.Em7.HmiInterface".cmJRWinderAxisB.configuration.setPositions[3].position, Maxipixel := 115, Minpixel :=, simHmiAxis => "Simulation".simHmiLinearAxis[21])
   END_RUNG
   // the same network as SCL:
   #"LER_SimAxis+_Axis05_pnp1X"(EN := #TRUE,   // "LER_SimAxis+"
                           axisActualPos := "Unit1.Em4.HmiInterface".cmAnodeMainPnP1AxisX.monitoring.actualPosition,
                           pixel := 760,
                           startposition := 0.0,
                           endposition := "Unit1.Em4.HmiInterface".cmAnodeMainPnP1AxisX.configuration.setPositions[0].position,
                           Maxipixel := 120,
                           Minpixel := 0,
                           simHmiAxis => "Simulation".simHmiLinearAxis[5],
                           ENO => #_w1);
   IF #_w1 THEN
       #"LER_SimAxis+_Axis12_pnp1Z"(axisActualPos := "Unit1.Em4.HmiInterface".cmAnodeMainPnP1AxisZ.monitoring.actualPosition,   // "LER_SimAxis+"
                               pixel := 234,
                               endposition := "Unit1.Em4.HmiInterface".cmAnodeMainPnP1AxisZ.configuration.setPositions[2].position,
                               Maxipixel := 100,
                               simHmiAxis => "Simulation".simHmiLinearAxis[12]);
   END_IF;
   #"LER_SimAxis+_Axis06_pnp2X"(EN := #TRUE,   // "LER_SimAxis+"
                           axisActualPos := "Unit1.Em4.HmiInterface".cmAnodeMainPnP2AxisX.monitoring.actualPosition,
                           pixel := 640,
                           startposition := 0.0,
                           endposition := "Unit1.Em4.HmiInterface".cmAnodeMainPnP2AxisX.configuration.setPositions[0].position,
                           Maxipixel := 120,
                           Minpixel := 0,
                           simHmiAxis => "Simulation".simHmiLinearAxis[6],
                           ENO => #_w2);
   IF #_w2 THEN
       #"LER_SimAxis+_Axis14_pnp2Z"(axisActualPos := "Unit1.Em4.HmiInterface".cmAnodeMainPnP2AxisZ.monitoring.actualPosition,   // "LER_SimAxis+"
                               pixel := 234,
                               startposition := 0.0,
                               endposition := "Unit1.Em4.HmiInterface".cmAnodeMainPnP2AxisZ.configuration.setPositions[2].position,
                               Maxipixel := 100,
                               simHmiAxis => "Simulation".simHmiLinearAxis[14]);
   END_IF;
   #"LER_SimAxis+_Axis07_pnp1X"(EN := #TRUE,   // "LER_SimAxis+"
                           axisActualPos := "Unit1.Em5.HmiInterface".cmCathodeMainPnP1AxisX.monitoring.actualPosition,
                           pixel := 400,
                           endposition := "Unit1.Em5.HmiInterface".cmCathodeMainPnP1AxisX.configuration.setPositions[2].position,
                           Maxipixel := 120,
                           Minpixel := 0,
                           simHmiAxis => "Simulation".simHmiLinearAxis[7],
                           ENO => #_w3);
   IF #_w3 THEN
       #"LER_SimAxis+_Axis10_pnp1Z"(axisActualPos := "Unit1.Em5.HmiInterface".cmCathodeMainPnP1AxisZ.monitoring.actualPosition,   // "LER_SimAxis+"
                               pixel := 234,
                               endposition := "Unit1.Em5.HmiInterface".cmCathodeMainPnP1AxisZ.configuration.setPositions[2].position,
                               Maxipixel := 100,
                               simHmiAxis => "Simulation".simHmiLinearAxis[10]);
   END_IF;
   #"LER_SimAxis+_Axis8_pnp2X"(EN := #TRUE,   // "LER_SimAxis+"
                           axisActualPos := "Unit1.Em5.HmiInterface".cmCathodeMainPnP2AxisX.monitoring.actualPosition,
                           pixel := 520,
                           startposition := 0.0,
                           endposition := "Unit1.Em5.HmiInterface".cmCathodeMainPnP2AxisX.configuration.setPositions[2].position,
                           Maxipixel := 120,
                           Minpixel := 0,
                           simHmiAxis => "Simulation".simHmiLinearAxis[8],
                           ENO => #_w4);
   IF #_w4 THEN
       #"LER_SimAxis+_Axis13_pnp2Z"(axisActualPos := "Unit1.Em5.HmiInterface".cmCathodeMainPnP2AxisZ.monitoring.actualPosition,   // "LER_SimAxis+"
                               pixel := 234,
                               startposition := 0.0,
                               endposition := "Unit1.Em5.HmiInterface".cmCathodeMainPnP2AxisZ.configuration.setPositions[2].position,
                               Maxipixel := 100,
                               simHmiAxis => "Simulation".simHmiLinearAxis[13]);
   END_IF;
   #"LER_SimAxis+_Axis34_cutterX"(EN := #TRUE,   // "LER_SimAxis+"
                           axisActualPos := "Unit1.Em7.HmiInterface".cmSepaClampnCutterAxisX.monitoring.actualPosition,
                           pixel := 718,
                           startposition := 0.0,
                           endposition := "Unit1.Em7.HmiInterface".cmSepaClampnCutterAxisX.configuration.setPositions[6].position,
                           Maxipixel := 200,
                           simHmiAxis => "Simulation".simHmiLinearAxis[34],
                           ENO => #_w5);
   #"LER_SimAxis+_Axis35_cutterZ"(EN := #_w5,   // "LER_SimAxis+"
                           axisActualPos := "Unit1.Em7.HmiInterface".cmSepaClampnCutterAxisZ.monitoring.actualPosition,
                           pixel := 46,
                           startposition := "Unit1.Em7.HmiInterface".cmSepaClampnCutterAxisZ.configuration.setPositions[3].position,
                           endposition := "Unit1.Em7.HmiInterface".cmSepaClampnCutterAxisZ.configuration.setPositions[1].position,
                           Maxipixel := 55,
                           simHmiAxis => "Simulation".simHmiLinearAxis[35],
                           ENO => #_w6);
   #"LER_SimAxis-_Axis36_GripperX"(EN := #_w6,   // "LER_SimAxis-"
                           axisActualPos := "Unit1.Em7.HmiInterface".cmSepaGripperAxisX.monitoring.actualPosition,
                           pixel := 1078,
                           endposition := "Unit1.Em7.HmiInterface".cmSepaGripperAxisX.configuration.setPositions[1].position,
                           Maxipixel := 250,
                           simHmiAxis => "Simulation".simHmiLinearAxis[36],
                           ENO => #_w7);
   IF #_w7 THEN
       #"LER_SimAxis+_Axis37_gripperZ"(axisActualPos := "Unit1.Em7.HmiInterface".cmSepaGripperAxisZ.monitoring.actualPosition,   // "LER_SimAxis+"
                               pixel := 28,
                               endposition := "Unit1.Em7.HmiInterface".cmSepaGripperAxisZ.configuration.setPositions[1].position,
                               Maxipixel := 55,
                               simHmiAxis => "Simulation".simHmiLinearAxis[37]);
   END_IF;
   #"LER_SimAxis-_Axis32_StackTableZ"(EN := #TRUE,   // "LER_SimAxis-"
                           axisActualPos := "Unit1.Em6.HmiInterface".cmStackTableOutFrontAxisZ.monitoring.actualPosition,
                           pixel := 312,
                           endposition := "Unit1.Em6.HmiInterface".cmStackTableOutFrontAxisZ.configuration.setPositions[1].position,
                           Maxipixel := 50,
                           simHmiAxis => "Simulation".simHmiLinearAxis[32],
                           ENO => #_w8);
   IF #_w8 THEN
       #"LER_SimAxis+_Axis21_roller"(axisActualPos := "Unit1.Em6.HmiInterface".cmFinalRollerFrontAxisX.monitoring.actualPosition,   // "LER_SimAxis+"
                               pixel := 585,
                               endposition := "Unit1.Em7.HmiInterface".cmJRWinderAxisB.configuration.setPositions[3].position,
                               Maxipixel := 115,
                               simHmiAxis => "Simulation".simHmiLinearAxis[21]);
   END_IF;
END_REGION

REGION Network 4: Simulation Rotary Axis
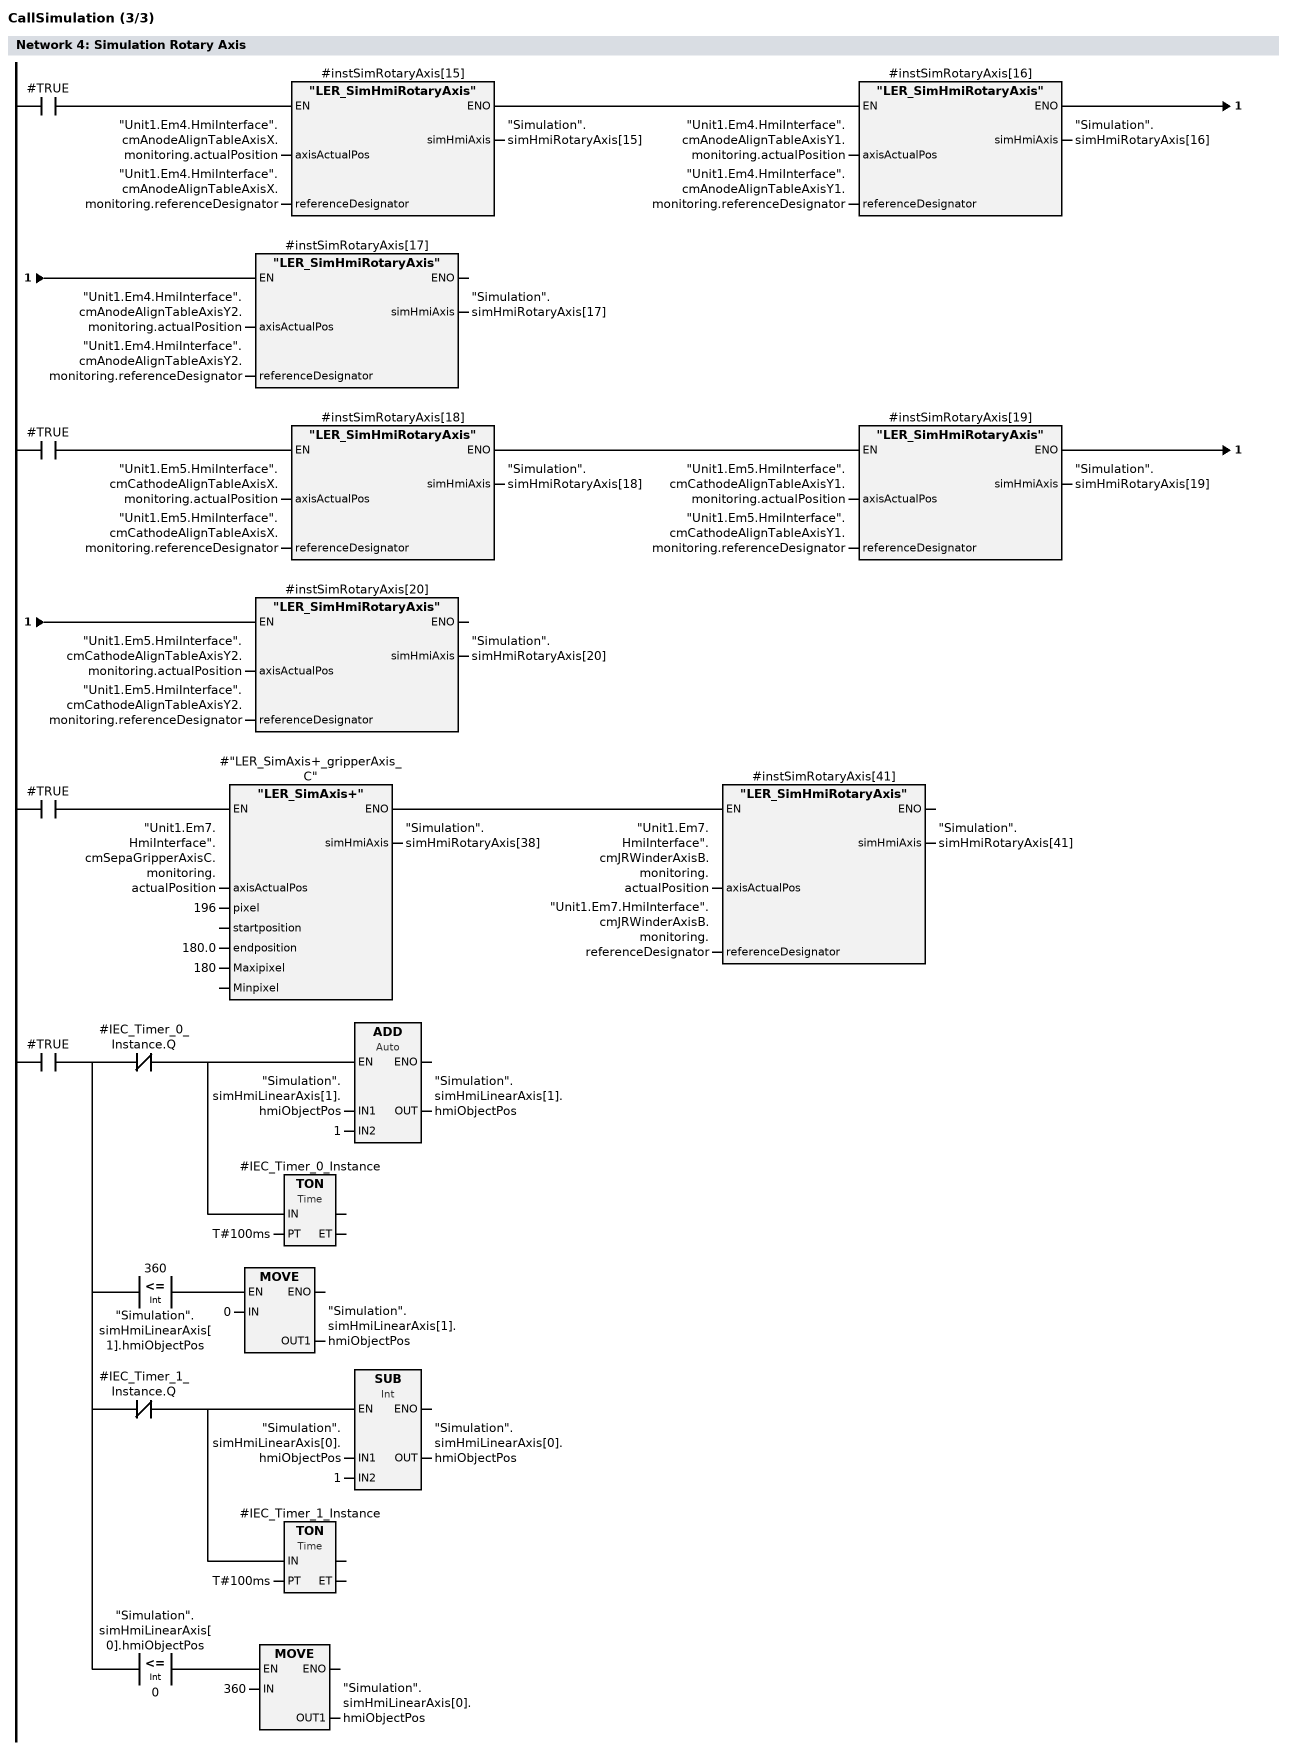
   RUNG wire#powerrail
      Contact( #TRUE )
      #instSimRotaryAxis[15](axisActualPos := "Unit1.Em4.HmiInterface".cmAnodeAlignTableAxisX.monitoring.actualPosition, referenceDesignator := "Unit1.Em4.HmiInterface".cmAnodeAlignTableAxisX.monitoring.referenceDesignator, simHmiAxis => "Simulation".simHmiRotaryAxis[15])
      #instSimRotaryAxis[16](axisActualPos := "Unit1.Em4.HmiInterface".cmAnodeAlignTableAxisY1.monitoring.actualPosition, referenceDesignator := "Unit1.Em4.HmiInterface".cmAnodeAlignTableAxisY1.monitoring.referenceDesignator, simHmiAxis => "Simulation".simHmiRotaryAxis[16])
      #instSimRotaryAxis[17](axisActualPos := "Unit1.Em4.HmiInterface".cmAnodeAlignTableAxisY2.monitoring.actualPosition, referenceDesignator := "Unit1.Em4.HmiInterface".cmAnodeAlignTableAxisY2.monitoring.referenceDesignator, simHmiAxis => "Simulation".simHmiRotaryAxis[17])
   END_RUNG
   RUNG wire#powerrail
      Contact( #TRUE )
      #instSimRotaryAxis[18](axisActualPos := "Unit1.Em5.HmiInterface".cmCathodeAlignTableAxisX.monitoring.actualPosition, referenceDesignator := "Unit1.Em5.HmiInterface".cmCathodeAlignTableAxisX.monitoring.referenceDesignator, simHmiAxis => "Simulation".simHmiRotaryAxis[18])
      #instSimRotaryAxis[19](axisActualPos := "Unit1.Em5.HmiInterface".cmCathodeAlignTableAxisY1.monitoring.actualPosition, referenceDesignator := "Unit1.Em5.HmiInterface".cmCathodeAlignTableAxisY1.monitoring.referenceDesignator, simHmiAxis => "Simulation".simHmiRotaryAxis[19])
      #instSimRotaryAxis[20](axisActualPos := "Unit1.Em5.HmiInterface".cmCathodeAlignTableAxisY2.monitoring.actualPosition, referenceDesignator := "Unit1.Em5.HmiInterface".cmCathodeAlignTableAxisY2.monitoring.referenceDesignator, simHmiAxis => "Simulation".simHmiRotaryAxis[20])
   END_RUNG
   RUNG wire#powerrail
      Contact( #TRUE )
      #"LER_SimAxis+_gripperAxis_C"(axisActualPos := "Unit1.Em7.HmiInterface".cmSepaGripperAxisC.monitoring.actualPosition, pixel := 196, startposition :=, endposition := 180.0, Maxipixel := 180, Minpixel :=, simHmiAxis => "Simulation".simHmiRotaryAxis[38])
      #instSimRotaryAxis[41](axisActualPos := "Unit1.Em7.HmiInterface".cmJRWinderAxisB.monitoring.actualPosition, referenceDesignator := "Unit1.Em7.HmiInterface".cmJRWinderAxisB.monitoring.referenceDesignator, simHmiAxis => "Simulation".simHmiRotaryAxis[41])
   END_RUNG
   RUNG wire#powerrail
      Contact( #TRUE )
      wire#w1
      I_Contact( #IEC_Timer_0_Instance.Q )
      wire#w2
      Add(in1 := "Simulation".simHmiLinearAxis[1].hmiObjectPos, in2 := 1, out => "Simulation".simHmiLinearAxis[1].hmiObjectPos)
   END_RUNG
   RUNG wire#w2
      { S7_Templates := "time_type := Time" } #IEC_Timer_0_Instance.TON(pt := T#100ms, et =>)
   END_RUNG
   RUNG wire#w1
      { S7_Templates := "SrcType := Int" } LE_Contact(in1 := 360, in2 := "Simulation".simHmiLinearAxis[1].hmiObjectPos)
      Move(in := 0, out1 => "Simulation".simHmiLinearAxis[1].hmiObjectPos)
   END_RUNG
   RUNG wire#w1
      I_Contact( #IEC_Timer_1_Instance.Q )
      wire#w3
      { S7_Templates := "SrcType := Int" } Sub(in1 := "Simulation".simHmiLinearAxis[0].hmiObjectPos, in2 := 1, out => "Simulation".simHmiLinearAxis[0].hmiObjectPos)
   END_RUNG
   RUNG wire#w3
      { S7_Templates := "time_type := Time" } #IEC_Timer_1_Instance.TON(pt := T#100ms, et =>)
   END_RUNG
   RUNG wire#w1
      { S7_Templates := "SrcType := Int" } LE_Contact(in1 := "Simulation".simHmiLinearAxis[0].hmiObjectPos, in2 := 0)
      Move(in := 360, out1 => "Simulation".simHmiLinearAxis[0].hmiObjectPos)
   END_RUNG
   // the same network as SCL:
   #instSimRotaryAxis[15](EN := #TRUE,   // "LER_SimHmiRotaryAxis"
                          axisActualPos := "Unit1.Em4.HmiInterface".cmAnodeAlignTableAxisX.monitoring.actualPosition,
                          referenceDesignator := "Unit1.Em4.HmiInterface".cmAnodeAlignTableAxisX.monitoring.referenceDesignator,
                          simHmiAxis => "Simulation".simHmiRotaryAxis[15],
                          ENO => #_w1);
   #instSimRotaryAxis[16](EN := #_w1,   // "LER_SimHmiRotaryAxis"
                          axisActualPos := "Unit1.Em4.HmiInterface".cmAnodeAlignTableAxisY1.monitoring.actualPosition,
                          referenceDesignator := "Unit1.Em4.HmiInterface".cmAnodeAlignTableAxisY1.monitoring.referenceDesignator,
                          simHmiAxis => "Simulation".simHmiRotaryAxis[16],
                          ENO => #_w2);
   IF #_w2 THEN
       #instSimRotaryAxis[17](axisActualPos := "Unit1.Em4.HmiInterface".cmAnodeAlignTableAxisY2.monitoring.actualPosition,   // "LER_SimHmiRotaryAxis"
                              referenceDesignator := "Unit1.Em4.HmiInterface".cmAnodeAlignTableAxisY2.monitoring.referenceDesignator,
                              simHmiAxis => "Simulation".simHmiRotaryAxis[17]);
   END_IF;
   #instSimRotaryAxis[18](EN := #TRUE,   // "LER_SimHmiRotaryAxis"
                          axisActualPos := "Unit1.Em5.HmiInterface".cmCathodeAlignTableAxisX.monitoring.actualPosition,
                          referenceDesignator := "Unit1.Em5.HmiInterface".cmCathodeAlignTableAxisX.monitoring.referenceDesignator,
                          simHmiAxis => "Simulation".simHmiRotaryAxis[18],
                          ENO => #_w3);
   #instSimRotaryAxis[19](EN := #_w3,   // "LER_SimHmiRotaryAxis"
                          axisActualPos := "Unit1.Em5.HmiInterface".cmCathodeAlignTableAxisY1.monitoring.actualPosition,
                          referenceDesignator := "Unit1.Em5.HmiInterface".cmCathodeAlignTableAxisY1.monitoring.referenceDesignator,
                          simHmiAxis => "Simulation".simHmiRotaryAxis[19],
                          ENO => #_w4);
   IF #_w4 THEN
       #instSimRotaryAxis[20](axisActualPos := "Unit1.Em5.HmiInterface".cmCathodeAlignTableAxisY2.monitoring.actualPosition,   // "LER_SimHmiRotaryAxis"
                              referenceDesignator := "Unit1.Em5.HmiInterface".cmCathodeAlignTableAxisY2.monitoring.referenceDesignator,
                              simHmiAxis => "Simulation".simHmiRotaryAxis[20]);
   END_IF;
   #"LER_SimAxis+_gripperAxis_C"(EN := #TRUE,   // "LER_SimAxis+"
                           axisActualPos := "Unit1.Em7.HmiInterface".cmSepaGripperAxisC.monitoring.actualPosition,
                           pixel := 196,
                           endposition := 180.0,
                           Maxipixel := 180,
                           simHmiAxis => "Simulation".simHmiRotaryAxis[38],
                           ENO => #_w5);
   IF #_w5 THEN
       #instSimRotaryAxis[41](axisActualPos := "Unit1.Em7.HmiInterface".cmJRWinderAxisB.monitoring.actualPosition,   // "LER_SimHmiRotaryAxis"
                              referenceDesignator := "Unit1.Em7.HmiInterface".cmJRWinderAxisB.monitoring.referenceDesignator,
                              simHmiAxis => "Simulation".simHmiRotaryAxis[41]);
   END_IF;
   #_w6 := #TRUE AND NOT #IEC_Timer_0_Instance.Q;
   IF #_w6 THEN
       "Simulation".simHmiLinearAxis[1].hmiObjectPos := "Simulation".simHmiLinearAxis[1].hmiObjectPos + 1;
   END_IF;
   #IEC_Timer_0_Instance(IN := #_w6, PT := T#100ms);   // TON
   IF #TRUE AND (360 <= "Simulation".simHmiLinearAxis[1].hmiObjectPos) THEN
       "Simulation".simHmiLinearAxis[1].hmiObjectPos := 0;
   END_IF;
   #_w7 := #TRUE AND NOT #IEC_Timer_1_Instance.Q;
   IF #_w7 THEN
       "Simulation".simHmiLinearAxis[0].hmiObjectPos := "Simulation".simHmiLinearAxis[0].hmiObjectPos - 1;
   END_IF;
   #IEC_Timer_1_Instance(IN := #_w7, PT := T#100ms);   // TON
   IF #TRUE AND ("Simulation".simHmiLinearAxis[0].hmiObjectPos <= 0) THEN
       "Simulation".simHmiLinearAxis[0].hmiObjectPos := 360;
   END_IF;
END_REGION
END_FUNCTION_BLOCK

FUNCTION "ParameterMove" : Void   // FC22, LAD
// stored: SetENOAutomatically false
   VAR_TEMP
      tempSoftCamDRApplyLoop : Array[1..41] of Int;
      tempSoftCamDRReadLoop : Array[1..41] of Int;
      tempButtonRisingEdge : "HMI_IF_Parameter_Save Button_UDT";
   END_VAR
   VAR_TEMP   // added for the SCL form of the ladder/FBD networks
      _w1 : Bool;
      _w2 : Bool;
      _w3 : Bool;
   END_VAR
BEGIN

REGION Network 2 (SCL): Button Rising Edge
   #tempButtonRisingEdge.Read := "HMI_Interface_Parameter"."Save Button".Read AND NOT "HMI_Interface_Parameter"."Save Button Old".Read;
   #tempButtonRisingEdge.Save := "HMI_Interface_Parameter"."Save Button".Save AND NOT "HMI_Interface_Parameter"."Save Button Old".Save;
   #tempButtonRisingEdge.Apply := "HMI_Interface_Parameter"."Save Button".Apply AND NOT "HMI_Interface_Parameter"."Save Button Old".Apply;
   "HMI_Interface_Parameter"."Save Button Old".Read := "HMI_Interface_Parameter"."Save Button".Read;
   "HMI_Interface_Parameter"."Save Button Old".Save := "HMI_Interface_Parameter"."Save Button".Save;
   "HMI_Interface_Parameter"."Save Button Old".Apply := "HMI_Interface_Parameter"."Save Button".Apply;
END_REGION

REGION Network 3 (SCL): HMI Parameter Text Set Value
   IF #tempButtonRisingEdge.Apply THEN
       "HMI_Interface_Parameter".Parameter_Text[0]."Process Value" := "HMI_Interface_Parameter".Parameter_Text[0]."Set Value";
       "HMI_Interface_Parameter".Parameter_Text[2]."Process Value" := "HMI_Interface_Parameter".Parameter_Text[2]."Set Value";
       "HMI_Interface_Parameter".Parameter_Text[6]."Process Value" := "HMI_Interface_Parameter".Parameter_Text[6]."Set Value";
       "HMI_Interface_Parameter".Parameter_Text[7]."Process Value" := "HMI_Interface_Parameter".Parameter_Text[7]."Set Value";
       "HMI_Interface_Parameter".Parameter_Text[9]."Process Value" := "HMI_Interface_Parameter".Parameter_Text[9]."Set Value";
       "HMI_Interface_Parameter".Parameter_Text[10]."Process Value" := "HMI_Interface_Parameter".Parameter_Text[10]."Set Value";
       "HMI_Interface_Parameter".Parameter_Text[11]."Process Value" := "HMI_Interface_Parameter".Parameter_Text[11]."Set Value";
       "HMI_Interface_Parameter".Parameter_Text[13]."Process Value" := "HMI_Interface_Parameter".Parameter_Text[13]."Set Value";
       "HMI_Interface_Parameter".Parameter_Text[14]."Process Value" := "HMI_Interface_Parameter".Parameter_Text[14]."Set Value";
       "HMI_Interface_Parameter".Parameter_Text[15]."Process Value" := "HMI_Interface_Parameter".Parameter_Text[15]."Set Value";
       "HMI_Interface_Parameter".Parameter_Text[16]."Process Value" := "HMI_Interface_Parameter".Parameter_Text[16]."Set Value";
       "HMI_Interface_Parameter".Parameter_Text[17]."Process Value" := "HMI_Interface_Parameter".Parameter_Text[17]."Set Value";
       "HMI_Interface_Parameter".Parameter_Text[18]."Process Value" := "HMI_Interface_Parameter".Parameter_Text[18]."Set Value";
       "HMI_Interface_Parameter".Parameter_Text[19]."Process Value" := "HMI_Interface_Parameter".Parameter_Text[19]."Set Value";
       "HMI_Interface_Parameter".Parameter_Text[20]."Process Value" := "HMI_Interface_Parameter".Parameter_Text[20]."Set Value";
       "HMI_Interface_Parameter".Parameter_Text[21]."Process Value" := "HMI_Interface_Parameter".Parameter_Text[21]."Set Value";
       "HMI_Interface_Parameter".Parameter_Text[22]."Process Value" := "HMI_Interface_Parameter".Parameter_Text[22]."Set Value";
       "HMI_Interface_Parameter".Parameter_Text[23]."Process Value" := "HMI_Interface_Parameter".Parameter_Text[23]."Set Value";
       "HMI_Interface_Parameter".Parameter_Text[24]."Process Value" := "HMI_Interface_Parameter".Parameter_Text[24]."Set Value";
       "HMI_Interface_Parameter".Parameter_Text[25]."Process Value" := "HMI_Interface_Parameter".Parameter_Text[25]."Set Value";
       "HMI_Interface_Parameter".Parameter_Text[26]."Process Value" := "HMI_Interface_Parameter".Parameter_Text[26]."Set Value";
       "HMI_Interface_Parameter".Parameter_Text[27]."Process Value" := "HMI_Interface_Parameter".Parameter_Text[27]."Set Value";
       "HMI_Interface_Parameter".Parameter_Text[28]."Process Value" := "HMI_Interface_Parameter".Parameter_Text[28]."Set Value";
       "HMI_Interface_Parameter".Parameter_Text[29]."Process Value" := "HMI_Interface_Parameter".Parameter_Text[29]."Set Value";
       "HMI_Interface_Parameter".Parameter_Text[30]."Process Value" := "HMI_Interface_Parameter".Parameter_Text[30]."Set Value";
       "HMI_Interface_Parameter".Parameter_Text[31]."Process Value" := "HMI_Interface_Parameter".Parameter_Text[31]."Set Value";
       "HMI_Interface_Parameter".Parameter_Text[32]."Process Value" := "HMI_Interface_Parameter".Parameter_Text[32]."Set Value";
       "HMI_Interface_Parameter".Parameter_Text[33]."Process Value" := "HMI_Interface_Parameter".Parameter_Text[33]."Set Value";
       "HMI_Interface_Parameter".Parameter_Text[34]."Process Value" := "HMI_Interface_Parameter".Parameter_Text[34]."Set Value";
       "HMI_Interface_Parameter".Parameter_Text[35]."Process Value" := "HMI_Interface_Parameter".Parameter_Text[35]."Set Value";
       "HMI_Interface_Parameter".Parameter_Text[36]."Process Value" := "HMI_Interface_Parameter".Parameter_Text[36]."Set Value";
       "HMI_Interface_Parameter".Parameter_Text[37]."Process Value" := "HMI_Interface_Parameter".Parameter_Text[37]."Set Value";
       "HMI_Interface_Parameter".Parameter_Text[38]."Process Value" := "HMI_Interface_Parameter".Parameter_Text[38]."Set Value";
       "HMI_Interface_Parameter".Parameter_Text[39]."Process Value" := "HMI_Interface_Parameter".Parameter_Text[39]."Set Value";
       "HMI_Interface_Parameter".Parameter_Text[40]."Process Value" := "HMI_Interface_Parameter".Parameter_Text[40]."Set Value";
       "HMI_Interface_Parameter".Parameter_Text[41]."Process Value" := "HMI_Interface_Parameter".Parameter_Text[41]."Set Value";
       "HMI_Interface_Parameter".Parameter_Text[42]."Process Value" := "HMI_Interface_Parameter".Parameter_Text[42]."Set Value";
       "HMI_Interface_Parameter".Parameter_Text[43]."Process Value" := "HMI_Interface_Parameter".Parameter_Text[43]."Set Value";
       "HMI_Interface_Parameter".Parameter_Text[44]."Process Value" := "HMI_Interface_Parameter".Parameter_Text[44]."Set Value";
       "HMI_Interface_Parameter".Parameter_Text[45]."Process Value" := "HMI_Interface_Parameter".Parameter_Text[45]."Set Value";
       "HMI_Interface_Parameter".Parameter_Text[46]."Process Value" := "HMI_Interface_Parameter".Parameter_Text[46]."Set Value";
       "HMI_Interface_Parameter".Parameter_Text[47]."Process Value" := "HMI_Interface_Parameter".Parameter_Text[47]."Set Value";
       "HMI_Interface_Parameter".Parameter_Text[48]."Process Value" := "HMI_Interface_Parameter".Parameter_Text[48]."Set Value";
       "HMI_Interface_Parameter".Parameter_Text[49]."Process Value" := "HMI_Interface_Parameter".Parameter_Text[49]."Set Value";
       "HMI_Interface_Parameter".Parameter_Text[50]."Process Value" := "HMI_Interface_Parameter".Parameter_Text[50]."Set Value";
       "HMI_Interface_Parameter".Parameter_Text[51]."Process Value" := "HMI_Interface_Parameter".Parameter_Text[51]."Set Value";
       "HMI_Interface_Parameter".Parameter_Text[52]."Process Value" := "HMI_Interface_Parameter".Parameter_Text[52]."Set Value";
       "HMI_Interface_Parameter".Parameter_Text[53]."Process Value" := "HMI_Interface_Parameter".Parameter_Text[53]."Set Value";
       "HMI_Interface_Parameter".Parameter_Text[54]."Process Value" := "HMI_Interface_Parameter".Parameter_Text[54]."Set Value";
       "HMI_Interface_Parameter".Parameter_Text[55]."Process Value" := "HMI_Interface_Parameter".Parameter_Text[55]."Set Value";
       "HMI_Interface_Parameter".Parameter_Text[56]."Process Value" := "HMI_Interface_Parameter".Parameter_Text[56]."Set Value";
       "HMI_Interface_Parameter".Parameter_Text[57]."Process Value" := "HMI_Interface_Parameter".Parameter_Text[57]."Set Value";
       "HMI_Interface_Parameter".Parameter_Text[58]."Process Value" := "HMI_Interface_Parameter".Parameter_Text[58]."Set Value";
       "HMI_Interface_Parameter".Parameter_Text[59]."Process Value" := "HMI_Interface_Parameter".Parameter_Text[59]."Set Value";
       "HMI_Interface_Parameter".Parameter_Text[60]."Process Value" := "HMI_Interface_Parameter".Parameter_Text[60]."Set Value";
       "HMI_Interface_Parameter".Parameter_Text[61]."Process Value" := "HMI_Interface_Parameter".Parameter_Text[61]."Set Value";
       "HMI_Interface_Parameter".Parameter_Text[62]."Process Value" := "HMI_Interface_Parameter".Parameter_Text[62]."Set Value";
       "HMI_Interface_Parameter".Parameter_Text[63]."Process Value" := "HMI_Interface_Parameter".Parameter_Text[63]."Set Value";
       "HMI_Interface_Parameter".Parameter_Text[64]."Process Value" := "HMI_Interface_Parameter".Parameter_Text[64]."Set Value";
       "HMI_Interface_Parameter".Parameter_Text[65]."Process Value" := "HMI_Interface_Parameter".Parameter_Text[65]."Set Value";
       "HMI_Interface_Parameter".Parameter_Text[66]."Process Value" := "HMI_Interface_Parameter".Parameter_Text[66]."Set Value";
       "HMI_Interface_Parameter".Parameter_Text[67]."Process Value" := "HMI_Interface_Parameter".Parameter_Text[67]."Set Value";
       "HMI_Interface_Parameter".Parameter_Text[68]."Process Value" := "HMI_Interface_Parameter".Parameter_Text[68]."Set Value";
       "HMI_Interface_Parameter".Parameter_Text[69]."Process Value" := "HMI_Interface_Parameter".Parameter_Text[69]."Set Value";
       "HMI_Interface_Parameter".Parameter_Text[70]."Process Value" := "HMI_Interface_Parameter".Parameter_Text[70]."Set Value";
       "HMI_Interface_Parameter".Parameter_Text[71]."Process Value" := "HMI_Interface_Parameter".Parameter_Text[71]."Set Value";
       "HMI_Interface_Parameter".Parameter_Text[72]."Process Value" := "HMI_Interface_Parameter".Parameter_Text[72]."Set Value";
       "HMI_Interface_Parameter".Parameter_Text[73]."Process Value" := "HMI_Interface_Parameter".Parameter_Text[73]."Set Value";
       "HMI_Interface_Parameter".Parameter_Text[74]."Process Value" := "HMI_Interface_Parameter".Parameter_Text[74]."Set Value";
       "HMI_Interface_Parameter".Parameter_Text[75]."Process Value" := "HMI_Interface_Parameter".Parameter_Text[75]."Set Value";
       "HMI_Interface_Parameter".Parameter_Text[76]."Process Value" := "HMI_Interface_Parameter".Parameter_Text[76]."Set Value";
       "HMI_Interface_Parameter".Parameter_Text[77]."Process Value" := "HMI_Interface_Parameter".Parameter_Text[77]."Set Value";
       "HMI_Interface_Parameter".Parameter_Text[78]."Process Value" := "HMI_Interface_Parameter".Parameter_Text[78]."Set Value";
       "HMI_Interface_Parameter".Parameter_Text[79]."Process Value" := "HMI_Interface_Parameter".Parameter_Text[79]."Set Value";
       "HMI_Interface_Parameter".Parameter_Text[80]."Process Value" := "HMI_Interface_Parameter".Parameter_Text[80]."Set Value";
       "HMI_Interface_Parameter".Parameter_Text[81]."Process Value" := "HMI_Interface_Parameter".Parameter_Text[81]."Set Value";
       "HMI_Interface_Parameter".Parameter_Text[82]."Process Value" := "HMI_Interface_Parameter".Parameter_Text[82]."Set Value";
       "HMI_Interface_Parameter".Parameter_Text[83]."Process Value" := "HMI_Interface_Parameter".Parameter_Text[83]."Set Value";
       "HMI_Interface_Parameter".Parameter_Text[84]."Process Value" := "HMI_Interface_Parameter".Parameter_Text[84]."Set Value";
       "HMI_Interface_Parameter".Parameter_Text[85]."Process Value" := "HMI_Interface_Parameter".Parameter_Text[85]."Set Value";
       "HMI_Interface_Parameter".Parameter_Text[86]."Process Value" := "HMI_Interface_Parameter".Parameter_Text[86]."Set Value";
       "HMI_Interface_Parameter".Parameter_Text[87]."Process Value" := "HMI_Interface_Parameter".Parameter_Text[87]."Set Value";
       "HMI_Interface_Parameter".Parameter_Text[88]."Process Value" := "HMI_Interface_Parameter".Parameter_Text[88]."Set Value";
       "HMI_Interface_Parameter".Parameter_Text[89]."Process Value" := "HMI_Interface_Parameter".Parameter_Text[89]."Set Value";
       "HMI_Interface_Parameter".Parameter_Text[90]."Process Value" := "HMI_Interface_Parameter".Parameter_Text[90]."Set Value";
       "HMI_Interface_Parameter".Parameter_Text[91]."Process Value" := "HMI_Interface_Parameter".Parameter_Text[91]."Set Value";
       "HMI_Interface_Parameter".Parameter_Text[92]."Process Value" := "HMI_Interface_Parameter".Parameter_Text[92]."Set Value";
       "HMI_Interface_Parameter".Parameter_Text[93]."Process Value" := "HMI_Interface_Parameter".Parameter_Text[93]."Set Value";
       "HMI_Interface_Parameter".Parameter_Text[94]."Process Value" := "HMI_Interface_Parameter".Parameter_Text[94]."Set Value";
       "HMI_Interface_Parameter".Parameter_Text[95]."Process Value" := "HMI_Interface_Parameter".Parameter_Text[95]."Set Value";
       "HMI_Interface_Parameter".Parameter_Text[96]."Process Value" := "HMI_Interface_Parameter".Parameter_Text[96]."Set Value";
       "HMI_Interface_Parameter".Parameter_Text[97]."Process Value" := "HMI_Interface_Parameter".Parameter_Text[97]."Set Value";
       "HMI_Interface_Parameter".Parameter_Text[98]."Process Value" := "HMI_Interface_Parameter".Parameter_Text[98]."Set Value";
       "HMI_Interface_Parameter".Parameter_Text[99]."Process Value" := "HMI_Interface_Parameter".Parameter_Text[99]."Set Value";
       "HMI_Interface_Parameter".Parameter_Text[100]."Process Value" := "HMI_Interface_Parameter".Parameter_Text[100]."Set Value";
       "HMI_Interface_Parameter".Parameter_Text[101]."Process Value" := "HMI_Interface_Parameter".Parameter_Text[101]."Set Value";
       "HMI_Interface_Parameter".Parameter_Text[102]."Process Value" := "HMI_Interface_Parameter".Parameter_Text[102]."Set Value";
       "HMI_Interface_Parameter".Parameter_Text[103]."Process Value" := "HMI_Interface_Parameter".Parameter_Text[103]."Set Value";
       "HMI_Interface_Parameter".Parameter_Text[104]."Process Value" := "HMI_Interface_Parameter".Parameter_Text[104]."Set Value";
       "HMI_Interface_Parameter".Parameter_Text[105]."Process Value" := "HMI_Interface_Parameter".Parameter_Text[105]."Set Value";
       "HMI_Interface_Parameter".Parameter_Text[106]."Process Value" := "HMI_Interface_Parameter".Parameter_Text[106]."Set Value";
       "HMI_Interface_Parameter".Parameter_Text[107]."Process Value" := "HMI_Interface_Parameter".Parameter_Text[107]."Set Value";
       "HMI_Interface_Parameter".Parameter_Text[108]."Process Value" := "HMI_Interface_Parameter".Parameter_Text[108]."Set Value";
       "HMI_Interface_Parameter".Parameter_Text[109]."Process Value" := "HMI_Interface_Parameter".Parameter_Text[109]."Set Value";
       "HMI_Interface_Parameter".Parameter_Text[110]."Process Value" := "HMI_Interface_Parameter".Parameter_Text[110]."Set Value";
       "HMI_Interface_Parameter".Parameter_Text[111]."Process Value" := "HMI_Interface_Parameter".Parameter_Text[111]."Set Value";
       "HMI_Interface_Parameter".Parameter_Text[112]."Process Value" := "HMI_Interface_Parameter".Parameter_Text[112]."Set Value";
       "HMI_Interface_Parameter".Parameter_Text[113]."Process Value" := "HMI_Interface_Parameter".Parameter_Text[113]."Set Value";
       "HMI_Interface_Parameter".Parameter_Text[114]."Process Value" := "HMI_Interface_Parameter".Parameter_Text[114]."Set Value";
       "HMI_Interface_Parameter".Parameter_Text[115]."Process Value" := "HMI_Interface_Parameter".Parameter_Text[115]."Set Value";
       "HMI_Interface_Parameter".Parameter_Text[116]."Process Value" := "HMI_Interface_Parameter".Parameter_Text[116]."Set Value";
       "HMI_Interface_Parameter".Parameter_Text[117]."Process Value" := "HMI_Interface_Parameter".Parameter_Text[117]."Set Value";
       "HMI_Interface_Parameter".Parameter_Text[118]."Process Value" := "HMI_Interface_Parameter".Parameter_Text[118]."Set Value";
       "HMI_Interface_Parameter".Parameter_Text[119]."Process Value" := "HMI_Interface_Parameter".Parameter_Text[119]."Set Value";
       "HMI_Interface_Parameter".Parameter_Text[120]."Process Value" := "HMI_Interface_Parameter".Parameter_Text[120]."Set Value";
       "HMI_Interface_Parameter".Parameter_Text[121]."Process Value" := "HMI_Interface_Parameter".Parameter_Text[121]."Set Value";
       "HMI_Interface_Parameter".Parameter_Text[122]."Process Value" := "HMI_Interface_Parameter".Parameter_Text[122]."Set Value";
       "HMI_Interface_Parameter".Parameter_Text[123]."Process Value" := "HMI_Interface_Parameter".Parameter_Text[123]."Set Value";
       "HMI_Interface_Parameter".Parameter_Text[124]."Process Value" := "HMI_Interface_Parameter".Parameter_Text[124]."Set Value";
       "HMI_Interface_Parameter".Parameter_Text[125]."Process Value" := "HMI_Interface_Parameter".Parameter_Text[125]."Set Value";
       "HMI_Interface_Parameter".Parameter_Text[126]."Process Value" := "HMI_Interface_Parameter".Parameter_Text[126]."Set Value";
       "HMI_Interface_Parameter".Parameter_Text[127]."Process Value" := "HMI_Interface_Parameter".Parameter_Text[127]."Set Value";
       "HMI_Interface_Parameter".Parameter_Text[128]."Process Value" := "HMI_Interface_Parameter".Parameter_Text[128]."Set Value";
       "HMI_Interface_Parameter".Parameter_Text[129]."Process Value" := "HMI_Interface_Parameter".Parameter_Text[129]."Set Value";
       "HMI_Interface_Parameter".Parameter_Text[130]."Process Value" := "HMI_Interface_Parameter".Parameter_Text[130]."Set Value";
       "HMI_Interface_Parameter".Parameter_Text[131]."Process Value" := "HMI_Interface_Parameter".Parameter_Text[131]."Set Value";
       "HMI_Interface_Parameter".Parameter_Text[132]."Process Value" := "HMI_Interface_Parameter".Parameter_Text[132]."Set Value";
       "HMI_Interface_Parameter".Parameter_Text[133]."Process Value" := "HMI_Interface_Parameter".Parameter_Text[133]."Set Value";
       "HMI_Interface_Parameter".Parameter_Text[134]."Process Value" := "HMI_Interface_Parameter".Parameter_Text[134]."Set Value";
       "HMI_Interface_Parameter".Parameter_Text[135]."Process Value" := "HMI_Interface_Parameter".Parameter_Text[135]."Set Value";
       "HMI_Interface_Parameter".Parameter_Text[136]."Process Value" := "HMI_Interface_Parameter".Parameter_Text[136]."Set Value";
       "HMI_Interface_Parameter".Parameter_Text[137]."Process Value" := "HMI_Interface_Parameter".Parameter_Text[137]."Set Value";
       "HMI_Interface_Parameter".Parameter_Text[138]."Process Value" := "HMI_Interface_Parameter".Parameter_Text[138]."Set Value";
       "HMI_Interface_Parameter".Parameter_Text[139]."Process Value" := "HMI_Interface_Parameter".Parameter_Text[139]."Set Value";
       "HMI_Interface_Parameter".Parameter_Text[140]."Process Value" := "HMI_Interface_Parameter".Parameter_Text[140]."Set Value";
       "HMI_Interface_Parameter".Parameter_Text[141]."Process Value" := "HMI_Interface_Parameter".Parameter_Text[141]."Set Value";
       "HMI_Interface_Parameter".Parameter_Text[142]."Process Value" := "HMI_Interface_Parameter".Parameter_Text[142]."Set Value";
       "HMI_Interface_Parameter".Parameter_Text[143]."Process Value" := "HMI_Interface_Parameter".Parameter_Text[143]."Set Value";
       "HMI_Interface_Parameter".Parameter_Text[144]."Process Value" := "HMI_Interface_Parameter".Parameter_Text[144]."Set Value";
       "HMI_Interface_Parameter".Parameter_Text[145]."Process Value" := "HMI_Interface_Parameter".Parameter_Text[145]."Set Value";
       "HMI_Interface_Parameter".Parameter_Text[146]."Process Value" := "HMI_Interface_Parameter".Parameter_Text[146]."Set Value";
       "HMI_Interface_Parameter".Parameter_Text[147]."Process Value" := "HMI_Interface_Parameter".Parameter_Text[147]."Set Value";
       "HMI_Interface_Parameter".Parameter_Text[148]."Process Value" := "HMI_Interface_Parameter".Parameter_Text[148]."Set Value";
       "HMI_Interface_Parameter".Parameter_Text[149]."Process Value" := "HMI_Interface_Parameter".Parameter_Text[149]."Set Value";
       "HMI_Interface_Parameter".Parameter_Text[150]."Process Value" := "HMI_Interface_Parameter".Parameter_Text[150]."Set Value";
       "HMI_Interface_Parameter".Parameter_Text[151]."Process Value" := "HMI_Interface_Parameter".Parameter_Text[151]."Set Value";
       "HMI_Interface_Parameter".Parameter_Text[152]."Process Value" := "HMI_Interface_Parameter".Parameter_Text[152]."Set Value";
       "HMI_Interface_Parameter".Parameter_Text[153]."Process Value" := "HMI_Interface_Parameter".Parameter_Text[153]."Set Value";
       "HMI_Interface_Parameter".Parameter_Text[154]."Process Value" := "HMI_Interface_Parameter".Parameter_Text[154]."Set Value";
   END_IF;
END_REGION

REGION Network 4 (SCL): HMI Parameter Image Set Value
   IF #tempButtonRisingEdge.Apply THEN
       // Move to recipe (Network 7)
       (* Unit1.Em3.HmiInterface.auxiliary.dancerRegulator := "HMI_Interface_Parameter".Parameter_Image[0]."Set Value";
       Unit1.Em0.HmiInterface.auxiliary.AutoSpliceRemainingLength := "HMI_Interface_Parameter".Parameter_Image[1]."Set Value";
       Unit1.Em1.HmiInterface.auxiliary.AutoSpliceRemainingLength := "HMI_Interface_Parameter".Parameter_Image[1]."Set Value"; *)
       "HMI_Interface_Parameter".FATModeInterface.HoursTest.ProcessValue.SelectHours_ProcessValue := "HMI_Interface_Parameter".FATModeInterface.HoursTest.SetValue.SelectHours_SetValue;
       "HMI_Interface_Parameter".FATModeInterface.Sampling.ProcessValue.SelectCount_ProcessValue := "HMI_Interface_Parameter".FATModeInterface.Sampling.SetValue.SelectCount_SetValue;
   END_IF;
   //
   //
   "Unit1.EmNodes".FATModeInterface.HoursTest.ProcessValue.SelectHours_ProcessValue := "HMI_Interface_Parameter".FATModeInterface.HoursTest.SetValue.SelectHours_SetValue;
   "Unit1.EmNodes".FATModeInterface.Sampling.ProcessValue.SelectCount_ProcessValue := "HMI_Interface_Parameter".FATModeInterface.Sampling.SetValue.SelectCount_SetValue;

   "HMI_Interface_Parameter".FATModeInterface.Capability.ProcessValue.CapabilityCount := LREAL_TO_INT("Unit1.EmNodes".BA060.InspectionToStack.InterfaceData.LReal[14]);
   "HMI_Interface_Parameter".FATModeInterface.Capability.ProcessValue.SelectCycle_ProcessValue := LREAL_TO_INT("Unit1.EmNodes".BA060.InspectionToStack.InterfaceData.LReal[15]);
   "HMI_Interface_Parameter".FATModeInterface.Capability.SetValue.SelectCycle_SetValue := LREAL_TO_INT("Unit1.EmNodes".BA060.InspectionToStack.InterfaceData.LReal[15]);


   "Unit1.EmNodes".FATModeInterface.Capability.ProcessValue.CapabilityCount := LREAL_TO_INT("Unit1.EmNodes".BA060.InspectionToStack.InterfaceData.LReal[14]);
   "Unit1.EmNodes".FATModeInterface.Capability.ProcessValue.SelectCycle_ProcessValue := LREAL_TO_INT("Unit1.EmNodes".BA060.InspectionToStack.InterfaceData.LReal[15]);
END_REGION

REGION Network 5 (SCL): HMI Parameter Text Process Value
   "Unit1.MotionNodes".PLCToMotion.Parameters.StackMain.Global.CPM := "HMI_Interface_Parameter".Parameter_Text[0]."Process Value";
   // FFU (Motion 소스 없음)
   // Unit1.MotionNodes.PLCToMotion.Parameters.StackMain.Auto.CellCount := LREAL_TO_DINT("HMI_Interface_Parameter".Parameter_Text[2]."Process Value");
   // JR Winding Turn Count (Motion 소스 없음)
   // Top Unwinder Bobin Size (Motion 소스 없음)
   // Bottom Unwinder Bobin Size (Motion 소스 없음)
   "Unit1.EmNodes".SleepModeActivationTime := DINT_TO_TIME(ROUND("HMI_Interface_Parameter".Parameter_Text[6]."Process Value" * 1000));
   "Unit1.EmNodes".DeepSleepModeActivationTime := DINT_TO_TIME(ROUND("HMI_Interface_Parameter".Parameter_Text[7]."Process Value" * 1000));
   // Reserve9 (Motion 소스 없음)
   "Unit1.MotionNodes".PLCToMotion.Parameters.Dancer.Setpoint := "HMI_Interface_Parameter".Parameter_Text[9]."Process Value";
   "Unit1.MotionNodes".PLCToMotion.Parameters.Dancer.Kp := "HMI_Interface_Parameter".Parameter_Text[10]."Process Value";
   "Unit1.MotionNodes".PLCToMotion.Parameters.Dancer.Ki := "HMI_Interface_Parameter".Parameter_Text[11]."Process Value";
   "Unit1.MotionNodes".PLCToMotion.Parameters.StackMain.Global.StageWidth := "HMI_Interface_Parameter".Parameter_Text[12]."Process Value";
   "Unit1.MotionNodes".PLCToMotion.Parameters.StackMain.Auto.Pos1FinalRollerXFwdOutputCam := "HMI_Interface_Parameter".Parameter_Text[13]."Process Value";
   "Unit1.MotionNodes".PLCToMotion.Parameters.StackMain.Auto.Pos1FinalRollerXBwdOutputCam := "HMI_Interface_Parameter".Parameter_Text[14]."Process Value";
   "Unit1.MotionNodes".PLCToMotion.Parameters.StackMain.Auto.Pos1FinalRollerXStackTableDownOutputCam := "HMI_Interface_Parameter".Parameter_Text[15]."Process Value";
   "Unit1.MotionNodes".PLCToMotion.Parameters.StackMain.Auto.Pos1FinalRollerXStackAnodeVisionOutputCam := "HMI_Interface_Parameter".Parameter_Text[16]."Process Value";
   "Unit1.MotionNodes".PLCToMotion.Parameters.StackMain.Auto.Pos1FinalRollerXStackCathodeVisionOutputCam := "HMI_Interface_Parameter".Parameter_Text[17]."Process Value";
   "Unit1.MotionNodes".PLCToMotion.Parameters.StackMain.Auto.Pos1AnodePnPX1FwdOutputCam := "HMI_Interface_Parameter".Parameter_Text[18]."Process Value";
   "Unit1.MotionNodes".PLCToMotion.Parameters.StackMain.Auto.Pos1AnodePnPX1BwdOutputCam := "HMI_Interface_Parameter".Parameter_Text[19]."Process Value";
   "Unit1.MotionNodes".PLCToMotion.Parameters.StackMain.Auto.Pos1AnodePnPX1ReelCutDataDeleteOffOutputCam := "HMI_Interface_Parameter".Parameter_Text[20]."Process Value";
   "Unit1.MotionNodes".PLCToMotion.Parameters.StackMain.Auto.Pos1AnodePnPX2FwdOutputCam := "HMI_Interface_Parameter".Parameter_Text[21]."Process Value";
   "Unit1.MotionNodes".PLCToMotion.Parameters.StackMain.Auto.Pos1AnodePnPX2BwdOutputCam := "HMI_Interface_Parameter".Parameter_Text[22]."Process Value";
   "Unit1.MotionNodes".PLCToMotion.Parameters.StackMain.Auto.Pos1AnodePnPZ1Down1OutputCam := "HMI_Interface_Parameter".Parameter_Text[23]."Process Value";
   "Unit1.MotionNodes".PLCToMotion.Parameters.StackMain.Auto.Pos1AnodePnPZ1Up1OutputCam := "HMI_Interface_Parameter".Parameter_Text[24]."Process Value";
   "Unit1.MotionNodes".PLCToMotion.Parameters.StackMain.Auto.Pos1AnodePnPZ2Down1OutputCam := "HMI_Interface_Parameter".Parameter_Text[25]."Process Value";
   "Unit1.MotionNodes".PLCToMotion.Parameters.StackMain.Auto.Pos1AnodePnPZ2Up1OutputCam := "HMI_Interface_Parameter".Parameter_Text[26]."Process Value";
   "Unit1.MotionNodes".PLCToMotion.Parameters.StackMain.Auto.Pos1AnodePnPZ1Down2OutputCam := "HMI_Interface_Parameter".Parameter_Text[27]."Process Value";
   "Unit1.MotionNodes".PLCToMotion.Parameters.StackMain.Auto.Pos1AnodePnPZ1Up2OutputCam := "HMI_Interface_Parameter".Parameter_Text[28]."Process Value";
   "Unit1.MotionNodes".PLCToMotion.Parameters.StackMain.Auto.Pos1AnodePnPZ2Down2OutputCam := "HMI_Interface_Parameter".Parameter_Text[29]."Process Value";
   "Unit1.MotionNodes".PLCToMotion.Parameters.StackMain.Auto.Pos1AnodePnPZ2Up2OutputCam := "HMI_Interface_Parameter".Parameter_Text[30]."Process Value";
   "Unit1.MotionNodes".PLCToMotion.Parameters.StackMain.Auto.Pos1AnodePnPZ1SuctionOnOutputCam := "HMI_Interface_Parameter".Parameter_Text[31]."Process Value";
   "Unit1.MotionNodes".PLCToMotion.Parameters.StackMain.Auto.Pos1AnodePnPZ1SuctionOffOutputCam := "HMI_Interface_Parameter".Parameter_Text[32]."Process Value";
   "Unit1.MotionNodes".PLCToMotion.Parameters.StackMain.Auto.Pos1AnodePnPZ1ReelCutBlowOutputCam := "HMI_Interface_Parameter".Parameter_Text[33]."Process Value";
   "Unit1.MotionNodes".PLCToMotion.Parameters.StackMain.Auto.Pos1AnodePnPZ1ReelCutDataDeleteOnOutputCam := "HMI_Interface_Parameter".Parameter_Text[34]."Process Value";
   "Unit1.MotionNodes".PLCToMotion.Parameters.StackMain.Auto.Pos1AnodePnPZ1AlignVisionOutputCam := "HMI_Interface_Parameter".Parameter_Text[35]."Process Value";
   "Unit1.MotionNodes".PLCToMotion.Parameters.StackMain.Auto.Pos1AnodePnPZ2SuctionOnOutputCam := "HMI_Interface_Parameter".Parameter_Text[36]."Process Value";
   "Unit1.MotionNodes".PLCToMotion.Parameters.StackMain.Auto.Pos1AnodePnPZ2SuctionOffOutputCam := "HMI_Interface_Parameter".Parameter_Text[37]."Process Value";
   "Unit1.MotionNodes".PLCToMotion.Parameters.StackMain.Auto.Pos1AnodeAlignSuctionOnOutputCam := "HMI_Interface_Parameter".Parameter_Text[38]."Process Value";
   "Unit1.MotionNodes".PLCToMotion.Parameters.StackMain.Auto.Pos1AnodeAlignSuctionOffOutputCam := "HMI_Interface_Parameter".Parameter_Text[39]."Process Value";
   "Unit1.MotionNodes".PLCToMotion.Parameters.StackMain.Auto.Pos1CathodePnPX1FwdOutputCam := "HMI_Interface_Parameter".Parameter_Text[40]."Process Value";
   "Unit1.MotionNodes".PLCToMotion.Parameters.StackMain.Auto.Pos1CathodePnPX1BwdOutputCam := "HMI_Interface_Parameter".Parameter_Text[41]."Process Value";
   "Unit1.MotionNodes".PLCToMotion.Parameters.StackMain.Auto.Pos1CathodePnPX1ReelCutDataDeleteOffOutputCam := "HMI_Interface_Parameter".Parameter_Text[42]."Process Value";
   "Unit1.MotionNodes".PLCToMotion.Parameters.StackMain.Auto.Pos1CathodePnPX2FwdOutputCam := "HMI_Interface_Parameter".Parameter_Text[43]."Process Value";
   "Unit1.MotionNodes".PLCToMotion.Parameters.StackMain.Auto.Pos1CathodePnPX2BwdOutputCam := "HMI_Interface_Parameter".Parameter_Text[44]."Process Value";
   "Unit1.MotionNodes".PLCToMotion.Parameters.StackMain.Auto.Pos1CathodePnPZ1Down1OutputCam := "HMI_Interface_Parameter".Parameter_Text[45]."Process Value";
   "Unit1.MotionNodes".PLCToMotion.Parameters.StackMain.Auto.Pos1CathodePnPZ1Up1OutputCam := "HMI_Interface_Parameter".Parameter_Text[46]."Process Value";
   "Unit1.MotionNodes".PLCToMotion.Parameters.StackMain.Auto.Pos1CathodePnPZ2Down1OutputCam := "HMI_Interface_Parameter".Parameter_Text[47]."Process Value";
   "Unit1.MotionNodes".PLCToMotion.Parameters.StackMain.Auto.Pos1CathodePnPZ2Up1OutputCam := "HMI_Interface_Parameter".Parameter_Text[48]."Process Value";
   "Unit1.MotionNodes".PLCToMotion.Parameters.StackMain.Auto.Pos1CathodePnPZ1Down2OutputCam := "HMI_Interface_Parameter".Parameter_Text[49]."Process Value";
   "Unit1.MotionNodes".PLCToMotion.Parameters.StackMain.Auto.Pos1CathodePnPZ1Up2OutputCam := "HMI_Interface_Parameter".Parameter_Text[50]."Process Value";
   "Unit1.MotionNodes".PLCToMotion.Parameters.StackMain.Auto.Pos1CathodePnPZ2Down2OutputCam := "HMI_Interface_Parameter".Parameter_Text[51]."Process Value";
   "Unit1.MotionNodes".PLCToMotion.Parameters.StackMain.Auto.Pos1CathodePnPZ2Up2OutputCam := "HMI_Interface_Parameter".Parameter_Text[52]."Process Value";
   "Unit1.MotionNodes".PLCToMotion.Parameters.StackMain.Auto.Pos1CathodePnPZ1SuctionOnOutputCam := "HMI_Interface_Parameter".Parameter_Text[53]."Process Value";
   "Unit1.MotionNodes".PLCToMotion.Parameters.StackMain.Auto.Pos1CathodePnPZ1SuctionOffOutputCam := "HMI_Interface_Parameter".Parameter_Text[54]."Process Value";
   "Unit1.MotionNodes".PLCToMotion.Parameters.StackMain.Auto.Pos1CathodePnPZ1ReelCutBlowOutputCam := "HMI_Interface_Parameter".Parameter_Text[55]."Process Value";
   "Unit1.MotionNodes".PLCToMotion.Parameters.StackMain.Auto.Pos1CathodePnPZ1ReelCutDataDeleteOnOutputCam := "HMI_Interface_Parameter".Parameter_Text[56]."Process Value";
   "Unit1.MotionNodes".PLCToMotion.Parameters.StackMain.Auto.Pos1CathodePnPZ1AlignVisionOutputCam := "HMI_Interface_Parameter".Parameter_Text[57]."Process Value";
   "Unit1.MotionNodes".PLCToMotion.Parameters.StackMain.Auto.Pos1CathodePnPZ2SuctionOnOutputCam := "HMI_Interface_Parameter".Parameter_Text[58]."Process Value";
   "Unit1.MotionNodes".PLCToMotion.Parameters.StackMain.Auto.Pos1CathodePnPZ2SuctionOffOutputCam := "HMI_Interface_Parameter".Parameter_Text[59]."Process Value";
   "Unit1.MotionNodes".PLCToMotion.Parameters.StackMain.Auto.Pos1CathodeAlignSuctionOnOutputCam := "HMI_Interface_Parameter".Parameter_Text[60]."Process Value";
   "Unit1.MotionNodes".PLCToMotion.Parameters.StackMain.Auto.Pos1CathodeAlignSuctionOffOutputCam := "HMI_Interface_Parameter".Parameter_Text[61]."Process Value";
   "Unit1.MotionNodes".PLCToMotion.Parameters.StackMain.Auto.Pos2FinalRollerXFwdOutputCam := "HMI_Interface_Parameter".Parameter_Text[62]."Process Value";
   "Unit1.MotionNodes".PLCToMotion.Parameters.StackMain.Auto.Pos2FinalRollerXBwdOutputCam := "HMI_Interface_Parameter".Parameter_Text[63]."Process Value";
   "Unit1.MotionNodes".PLCToMotion.Parameters.StackMain.Auto.Pos2FinalRollerXStackTableDownOutputCam := "HMI_Interface_Parameter".Parameter_Text[64]."Process Value";
   "Unit1.MotionNodes".PLCToMotion.Parameters.StackMain.Auto.Pos2FinalRollerXStackAnodeVisionOutputCam := "HMI_Interface_Parameter".Parameter_Text[65]."Process Value";
   "Unit1.MotionNodes".PLCToMotion.Parameters.StackMain.Auto.Pos2FinalRollerXStackCathodeVisionOutputCam := "HMI_Interface_Parameter".Parameter_Text[66]."Process Value";
   "Unit1.MotionNodes".PLCToMotion.Parameters.StackMain.Auto.Pos2AnodePnPX1FwdOutputCam := "HMI_Interface_Parameter".Parameter_Text[67]."Process Value";
   "Unit1.MotionNodes".PLCToMotion.Parameters.StackMain.Auto.Pos2AnodePnPX1BwdOutputCam := "HMI_Interface_Parameter".Parameter_Text[68]."Process Value";
   "Unit1.MotionNodes".PLCToMotion.Parameters.StackMain.Auto.Pos2AnodePnPX1ReelCutDataDeleteOffOutputCam := "HMI_Interface_Parameter".Parameter_Text[69]."Process Value";
   "Unit1.MotionNodes".PLCToMotion.Parameters.StackMain.Auto.Pos2AnodePnPX2FwdOutputCam := "HMI_Interface_Parameter".Parameter_Text[70]."Process Value";
   "Unit1.MotionNodes".PLCToMotion.Parameters.StackMain.Auto.Pos2AnodePnPX2BwdOutputCam := "HMI_Interface_Parameter".Parameter_Text[71]."Process Value";
   "Unit1.MotionNodes".PLCToMotion.Parameters.StackMain.Auto.Pos2AnodePnPZ1Down1OutputCam := "HMI_Interface_Parameter".Parameter_Text[72]."Process Value";
   "Unit1.MotionNodes".PLCToMotion.Parameters.StackMain.Auto.Pos2AnodePnPZ1Up1OutputCam := "HMI_Interface_Parameter".Parameter_Text[73]."Process Value";
   "Unit1.MotionNodes".PLCToMotion.Parameters.StackMain.Auto.Pos2AnodePnPZ2Down1OutputCam := "HMI_Interface_Parameter".Parameter_Text[74]."Process Value";
   "Unit1.MotionNodes".PLCToMotion.Parameters.StackMain.Auto.Pos2AnodePnPZ2Up1OutputCam := "HMI_Interface_Parameter".Parameter_Text[75]."Process Value";
   "Unit1.MotionNodes".PLCToMotion.Parameters.StackMain.Auto.Pos2AnodePnPZ1Down2OutputCam := "HMI_Interface_Parameter".Parameter_Text[76]."Process Value";
   "Unit1.MotionNodes".PLCToMotion.Parameters.StackMain.Auto.Pos2AnodePnPZ1Up2OutputCam := "HMI_Interface_Parameter".Parameter_Text[77]."Process Value";
   "Unit1.MotionNodes".PLCToMotion.Parameters.StackMain.Auto.Pos2AnodePnPZ2Down2OutputCam := "HMI_Interface_Parameter".Parameter_Text[78]."Process Value";
   "Unit1.MotionNodes".PLCToMotion.Parameters.StackMain.Auto.Pos2AnodePnPZ2Up2OutputCam := "HMI_Interface_Parameter".Parameter_Text[79]."Process Value";
   "Unit1.MotionNodes".PLCToMotion.Parameters.StackMain.Auto.Pos2AnodePnPZ1SuctionOnOutputCam := "HMI_Interface_Parameter".Parameter_Text[80]."Process Value";
   "Unit1.MotionNodes".PLCToMotion.Parameters.StackMain.Auto.Pos2AnodePnPZ1SuctionOffOutputCam := "HMI_Interface_Parameter".Parameter_Text[81]."Process Value";
   "Unit1.MotionNodes".PLCToMotion.Parameters.StackMain.Auto.Pos2AnodePnPZ1ReelCutBlowOutputCam := "HMI_Interface_Parameter".Parameter_Text[82]."Process Value";
   "Unit1.MotionNodes".PLCToMotion.Parameters.StackMain.Auto.Pos2AnodePnPZ1ReelCutDataDeleteOnOutputCam := "HMI_Interface_Parameter".Parameter_Text[83]."Process Value";
   "Unit1.MotionNodes".PLCToMotion.Parameters.StackMain.Auto.Pos2AnodePnPZ1AlignVisionOutputCam := "HMI_Interface_Parameter".Parameter_Text[84]."Process Value";
   "Unit1.MotionNodes".PLCToMotion.Parameters.StackMain.Auto.Pos2AnodePnPZ2SuctionOnOutputCam := "HMI_Interface_Parameter".Parameter_Text[85]."Process Value";
   "Unit1.MotionNodes".PLCToMotion.Parameters.StackMain.Auto.Pos2AnodePnPZ2SuctionOffOutputCam := "HMI_Interface_Parameter".Parameter_Text[86]."Process Value";
   "Unit1.MotionNodes".PLCToMotion.Parameters.StackMain.Auto.Pos2AnodeAlignSuctionOnOutputCam := "HMI_Interface_Parameter".Parameter_Text[87]."Process Value";
   "Unit1.MotionNodes".PLCToMotion.Parameters.StackMain.Auto.Pos2AnodeAlignSuctionOffOutputCam := "HMI_Interface_Parameter".Parameter_Text[88]."Process Value";
   "Unit1.MotionNodes".PLCToMotion.Parameters.StackMain.Auto.Pos2CathodePnPX1FwdOutputCam := "HMI_Interface_Parameter".Parameter_Text[89]."Process Value";
   "Unit1.MotionNodes".PLCToMotion.Parameters.StackMain.Auto.Pos2CathodePnPX1BwdOutputCam := "HMI_Interface_Parameter".Parameter_Text[90]."Process Value";
   "Unit1.MotionNodes".PLCToMotion.Parameters.StackMain.Auto.Pos2CathodePnPX1ReelCutDataDeleteOffOutputCam := "HMI_Interface_Parameter".Parameter_Text[91]."Process Value";
   "Unit1.MotionNodes".PLCToMotion.Parameters.StackMain.Auto.Pos2CathodePnPX2FwdOutputCam := "HMI_Interface_Parameter".Parameter_Text[92]."Process Value";
   "Unit1.MotionNodes".PLCToMotion.Parameters.StackMain.Auto.Pos2CathodePnPX2BwdOutputCam := "HMI_Interface_Parameter".Parameter_Text[93]."Process Value";
   "Unit1.MotionNodes".PLCToMotion.Parameters.StackMain.Auto.Pos2CathodePnPZ1Down1OutputCam := "HMI_Interface_Parameter".Parameter_Text[94]."Process Value";
   "Unit1.MotionNodes".PLCToMotion.Parameters.StackMain.Auto.Pos2CathodePnPZ1Up1OutputCam := "HMI_Interface_Parameter".Parameter_Text[95]."Process Value";
   "Unit1.MotionNodes".PLCToMotion.Parameters.StackMain.Auto.Pos2CathodePnPZ2Down1OutputCam := "HMI_Interface_Parameter".Parameter_Text[96]."Process Value";
   "Unit1.MotionNodes".PLCToMotion.Parameters.StackMain.Auto.Pos2CathodePnPZ2Up1OutputCam := "HMI_Interface_Parameter".Parameter_Text[97]."Process Value";
   "Unit1.MotionNodes".PLCToMotion.Parameters.StackMain.Auto.Pos2CathodePnPZ1Down2OutputCam := "HMI_Interface_Parameter".Parameter_Text[98]."Process Value";
   "Unit1.MotionNodes".PLCToMotion.Parameters.StackMain.Auto.Pos2CathodePnPZ1Up2OutputCam := "HMI_Interface_Parameter".Parameter_Text[99]."Process Value";
   "Unit1.MotionNodes".PLCToMotion.Parameters.StackMain.Auto.Pos2CathodePnPZ2Down2OutputCam := "HMI_Interface_Parameter".Parameter_Text[100]."Process Value";
   "Unit1.MotionNodes".PLCToMotion.Parameters.StackMain.Auto.Pos2CathodePnPZ2Up2OutputCam := "HMI_Interface_Parameter".Parameter_Text[101]."Process Value";
   "Unit1.MotionNodes".PLCToMotion.Parameters.StackMain.Auto.Pos2CathodePnPZ1SuctionOnOutputCam := "HMI_Interface_Parameter".Parameter_Text[102]."Process Value";
   "Unit1.MotionNodes".PLCToMotion.Parameters.StackMain.Auto.Pos2CathodePnPZ1SuctionOffOutputCam := "HMI_Interface_Parameter".Parameter_Text[103]."Process Value";
   "Unit1.MotionNodes".PLCToMotion.Parameters.StackMain.Auto.Pos2CathodePnPZ1ReelCutBlowOutputCam := "HMI_Interface_Parameter".Parameter_Text[104]."Process Value";
   "Unit1.MotionNodes".PLCToMotion.Parameters.StackMain.Auto.Pos2CathodePnPZ1ReelCutDataDeleteOnOutputCam := "HMI_Interface_Parameter".Parameter_Text[105]."Process Value";
   "Unit1.MotionNodes".PLCToMotion.Parameters.StackMain.Auto.Pos2CathodePnPZ1AlignVisionOutputCam := "HMI_Interface_Parameter".Parameter_Text[106]."Process Value";
   "Unit1.MotionNodes".PLCToMotion.Parameters.StackMain.Auto.Pos2CathodePnPZ2SuctionOnOutputCam := "HMI_Interface_Parameter".Parameter_Text[107]."Process Value";
   "Unit1.MotionNodes".PLCToMotion.Parameters.StackMain.Auto.Pos2CathodePnPZ2SuctionOffOutputCam := "HMI_Interface_Parameter".Parameter_Text[108]."Process Value";
   "Unit1.MotionNodes".PLCToMotion.Parameters.StackMain.Auto.Pos2CathodeAlignSuctionOnOutputCam := "HMI_Interface_Parameter".Parameter_Text[109]."Process Value";
   "Unit1.MotionNodes".PLCToMotion.Parameters.StackMain.Auto.Pos2CathodeAlignSuctionOffOutputCam := "HMI_Interface_Parameter".Parameter_Text[110]."Process Value";
   "Unit1.MotionNodes".PLCToMotion.Parameters.StackMain.StackCalculate.StageHeight := "HMI_Interface_Parameter".Parameter_Text[111]."Process Value";
   "Unit1.MotionNodes".PLCToMotion.Parameters.StackMain.StackCalculate.StageGap := "HMI_Interface_Parameter".Parameter_Text[112]."Process Value";
   "Unit1.MotionNodes".PLCToMotion.Parameters.StackMain.StackCalculate.Ratio.FinalRollerStart := "HMI_Interface_Parameter".Parameter_Text[113]."Process Value";
   "Unit1.MotionNodes".PLCToMotion.Parameters.StackMain.StackCalculate.Ratio.FinalRollerEnd := "HMI_Interface_Parameter".Parameter_Text[114]."Process Value";
   "Unit1.MotionNodes".PLCToMotion.Parameters.StackMain.StackCalculate.Ratio.PnPXStart := "HMI_Interface_Parameter".Parameter_Text[115]."Process Value";
   "Unit1.MotionNodes".PLCToMotion.Parameters.StackMain.StackCalculate.Ratio.PnPXEnd := "HMI_Interface_Parameter".Parameter_Text[116]."Process Value";
   "Unit1.MotionNodes".PLCToMotion.Parameters.StackMain.StackCalculate.Ratio.PnPZDownStart := "HMI_Interface_Parameter".Parameter_Text[117]."Process Value";
   "Unit1.MotionNodes".PLCToMotion.Parameters.StackMain.StackCalculate.Ratio.PnPZDownEnd := "HMI_Interface_Parameter".Parameter_Text[118]."Process Value";
   "Unit1.MotionNodes".PLCToMotion.Parameters.StackMain.StackCalculate.Ratio.PnPZUpStart := "HMI_Interface_Parameter".Parameter_Text[119]."Process Value";
   "Unit1.MotionNodes".PLCToMotion.Parameters.StackMain.StackCalculate.Ratio.PnPZUpEnd := "HMI_Interface_Parameter".Parameter_Text[120]."Process Value";
   "Unit1.MotionNodes".PLCToMotion.Parameters.StackMain.StackCalculate.Ratio.MandrelBwdStart := "HMI_Interface_Parameter".Parameter_Text[121]."Process Value";
   "Unit1.MotionNodes".PLCToMotion.Parameters.StackMain.StackCalculate.Ratio.MandrelBwdEnd := "HMI_Interface_Parameter".Parameter_Text[122]."Process Value";
   "Unit1.MotionNodes".PLCToMotion.Parameters.StackMain.StackCalculate.Ratio.MandrelFwdStart := "HMI_Interface_Parameter".Parameter_Text[123]."Process Value";
   "Unit1.MotionNodes".PLCToMotion.Parameters.StackMain.StackCalculate.Ratio.MandrelFwdEnd := "HMI_Interface_Parameter".Parameter_Text[124]."Process Value";
   "Unit1.MotionNodes".PLCToMotion.Parameters.StackMain.StackCalculate.Ratio.MandrelUpStart1 := "HMI_Interface_Parameter".Parameter_Text[125]."Process Value";
   "Unit1.MotionNodes".PLCToMotion.Parameters.StackMain.StackCalculate.Ratio.MandrelUpEnd1 := "HMI_Interface_Parameter".Parameter_Text[126]."Process Value";
   "Unit1.MotionNodes".PLCToMotion.Parameters.StackMain.StackCalculate.Ratio.MandrelUpStart2 := "HMI_Interface_Parameter".Parameter_Text[127]."Process Value";
   "Unit1.MotionNodes".PLCToMotion.Parameters.StackMain.StackCalculate.Ratio.MandrelUpEnd2 := "HMI_Interface_Parameter".Parameter_Text[128]."Process Value";
   "Unit1.MotionNodes".PLCToMotion.Parameters.StackMain.StackCalculate.Ratio.MandrelDownStart := "HMI_Interface_Parameter".Parameter_Text[129]."Process Value";
   "Unit1.MotionNodes".PLCToMotion.Parameters.StackMain.StackCalculate.Ratio.MandrelDownEnd := "HMI_Interface_Parameter".Parameter_Text[130]."Process Value";
   "Unit1.MotionNodes".PLCToMotion.Parameters.StackMain.StackCalculate.Ratio.MandrelYTerm := "HMI_Interface_Parameter".Parameter_Text[131]."Process Value";
   "Unit1.MotionNodes".PLCToMotion.Parameters.StackMain.StackCalculate.Ratio.MandrelZTerm := "HMI_Interface_Parameter".Parameter_Text[132]."Process Value";
   "Unit1.MotionNodes".PLCToMotion.Parameters.StackMain.StackCalculate.Ratio.MandrelBwdOffset := "HMI_Interface_Parameter".Parameter_Text[133]."Process Value";
   "Unit1.MotionNodes".PLCToMotion.Parameters.StackMain.StackCalculate.Ratio.MandrelFwdOffset := "HMI_Interface_Parameter".Parameter_Text[134]."Process Value";
   "Unit1.MotionNodes".PLCToMotion.Parameters.StackMain.StackCalculate.Time.FinalRollerStart := "HMI_Interface_Parameter".Parameter_Text[135]."Process Value";
   "Unit1.MotionNodes".PLCToMotion.Parameters.StackMain.StackCalculate.Time.FinalRollerEnd := "HMI_Interface_Parameter".Parameter_Text[136]."Process Value";
   "Unit1.MotionNodes".PLCToMotion.Parameters.StackMain.StackCalculate.Time.PnPXStart := "HMI_Interface_Parameter".Parameter_Text[137]."Process Value";
   "Unit1.MotionNodes".PLCToMotion.Parameters.StackMain.StackCalculate.Time.PnPXEnd := "HMI_Interface_Parameter".Parameter_Text[138]."Process Value";
   "Unit1.MotionNodes".PLCToMotion.Parameters.StackMain.StackCalculate.Time.PnPZDownStart := "HMI_Interface_Parameter".Parameter_Text[139]."Process Value";
   "Unit1.MotionNodes".PLCToMotion.Parameters.StackMain.StackCalculate.Time.PnPZDownEnd := "HMI_Interface_Parameter".Parameter_Text[140]."Process Value";
   "Unit1.MotionNodes".PLCToMotion.Parameters.StackMain.StackCalculate.Time.PnPZUpStart := "HMI_Interface_Parameter".Parameter_Text[141]."Process Value";
   "Unit1.MotionNodes".PLCToMotion.Parameters.StackMain.StackCalculate.Time.PnPZUpEnd := "HMI_Interface_Parameter".Parameter_Text[142]."Process Value";
   "Unit1.MotionNodes".PLCToMotion.Parameters.StackMain.StackCalculate.Time.MandrelBwdStart := "HMI_Interface_Parameter".Parameter_Text[143]."Process Value";
   "Unit1.MotionNodes".PLCToMotion.Parameters.StackMain.StackCalculate.Time.MandrelBwdEnd := "HMI_Interface_Parameter".Parameter_Text[144]."Process Value";
   "Unit1.MotionNodes".PLCToMotion.Parameters.StackMain.StackCalculate.Time.MandrelFwdStart := "HMI_Interface_Parameter".Parameter_Text[145]."Process Value";
   "Unit1.MotionNodes".PLCToMotion.Parameters.StackMain.StackCalculate.Time.MandrelFwdEnd := "HMI_Interface_Parameter".Parameter_Text[146]."Process Value";
   "Unit1.MotionNodes".PLCToMotion.Parameters.StackMain.StackCalculate.Time.MandrelUpStart1 := "HMI_Interface_Parameter".Parameter_Text[147]."Process Value";
   "Unit1.MotionNodes".PLCToMotion.Parameters.StackMain.StackCalculate.Time.MandrelUpEnd1 := "HMI_Interface_Parameter".Parameter_Text[148]."Process Value";
   "Unit1.MotionNodes".PLCToMotion.Parameters.StackMain.StackCalculate.Time.MandrelUpStart2 := "HMI_Interface_Parameter".Parameter_Text[149]."Process Value";
   "Unit1.MotionNodes".PLCToMotion.Parameters.StackMain.StackCalculate.Time.MandrelUpEnd2 := "HMI_Interface_Parameter".Parameter_Text[150]."Process Value";
   "Unit1.MotionNodes".PLCToMotion.Parameters.StackMain.StackCalculate.Time.MandrelDownStart := "HMI_Interface_Parameter".Parameter_Text[151]."Process Value";
   "Unit1.MotionNodes".PLCToMotion.Parameters.StackMain.StackCalculate.Time.MandrelDownEnd := "HMI_Interface_Parameter".Parameter_Text[152]."Process Value";
   "Unit1.MotionNodes".PLCToMotion.Parameters.StackMain.StackCalculate.Position.FinalRollerBwdPos := "HMI_Interface_Parameter".Parameter_Text[153]."Process Value";
   "Unit1.MotionNodes".PLCToMotion.Parameters.StackMain.StackCalculate.Position.FinalRollerFwdPos := "HMI_Interface_Parameter".Parameter_Text[154]."Process Value";
END_REGION

REGION Network 6 (SCL): HMI Parameter Image Process Value
   // Move to recipe (Network 7)
   //"HMI_Interface_Parameter".Parameter_Image[0]."Process Value" := Unit1.Em3.HmiInterface.auxiliary.dancerRegulator;
   //"HMI_Interface_Parameter".Parameter_Image[1]."Process Value" := Unit1.Em0.HmiInterface.auxiliary.AutoSpliceRemainingLength;
   //
   //"HMI_Interface_Parameter".Parameter_Image[1]."Process Value" := Unit1.Em1.HmiInterface.auxiliary.AutoSpliceRemainingLength;
END_REGION

REGION Network 7 (SCL): PLC -> Motion Teaching Start / End Pos (YS)
   /// Start Pos
   //
   "Unit1.MotionNodes".PLCToMotion.Parameters.StackMain.StackCalculate.TeachingPos.StartPos.Compensator := "Unit1.Em3.Config".cmCompensatorAxisX.setPositions[0].position;
   "Unit1.MotionNodes".PLCToMotion.Parameters.StackMain.StackCalculate.TeachingPos.StartPos.FinalRoller := "Unit1.Em6.Config".cmFinalRollerFrontAxisX.setPositions[0].position;

   "Unit1.MotionNodes".PLCToMotion.Parameters.StackMain.StackCalculate.TeachingPos.StartPos.AnodePnPX1 := "Unit1.Em4.Config".cmAnodeMainPnP1AxisX.setPositions[0].position;
   "Unit1.MotionNodes".PLCToMotion.Parameters.StackMain.StackCalculate.TeachingPos.StartPos.AnodePnPX2 := "Unit1.Em4.Config".cmAnodeMainPnP2AxisX.setPositions[0].position;
   "Unit1.MotionNodes".PLCToMotion.Parameters.StackMain.StackCalculate.TeachingPos.StartPos.AnodePnPZ1 := "Unit1.Em4.Config".cmAnodeMainPnP1AxisZ.setPositions[0].position;
   "Unit1.MotionNodes".PLCToMotion.Parameters.StackMain.StackCalculate.TeachingPos.StartPos.AnodePnPZ2 := "Unit1.Em4.Config".cmAnodeMainPnP2AxisZ.setPositions[0].position;

